ht_CAN4_ADDB_Tx.ID		:=	16#18200BDD OR EPEC_CANVXD.MASK_29BIT;
ht_CAN4_ADDB_Tx.Data[0]	:=	OrionBMS2_Rx.OrionBMS2_6BB_Rx.au8_Data[0];
ht_CAN4_ADDB_Tx.Data[1]	:=	OrionBMS2_Rx.OrionBMS2_6BB_Rx.au8_Data[1];
ht_CAN4_ADDB_Tx.Data[2]	:=	OrionBMS2_Rx.OrionBMS2_6BB_Rx.au8_Data[2];
ht_CAN4_ADDB_Tx.Data[3]	:=	OrionBMS2_Rx.OrionBMS2_6BB_Rx.au8_Data[3];
ht_CAN4_ADDB_Tx.Data[4]	:=	OrionBMS2_Rx.OrionBMS2_6BB_Rx.au8_Data[4];
ht_CAN4_ADDB_Tx.Data[5]	:=	OrionBMS2_Rx.OrionBMS2_6BB_Rx.au8_Data[5];		
ht_CAN4_ADDB_Tx.Data[6]	:=	OrionBMS2_Rx.OrionBMS2_6BB_Rx.au8_Data[6];	
ht_CAN4_ADDB_Tx.Data[7]	:=	OrionBMS2_Rx.OrionBMS2_6BB_Rx.au8_Data[7];		
ht_CAN4_ADDB_Tx.Len		:=	8;

ht_CAN4_ADDC_Tx.ID		:=	16#18200CDD OR EPEC_CANVXD.MASK_29BIT;
ht_CAN4_ADDC_Tx.Data[0]	:=	OrionBMS2_Rx.OrionBMS2_6BC_Rx.au8_Data[0];
ht_CAN4_ADDC_Tx.Data[1]	:=	OrionBMS2_Rx.OrionBMS2_6BC_Rx.au8_Data[1];
ht_CAN4_ADDC_Tx.Data[2]	:=	OrionBMS2_Rx.OrionBMS2_6BC_Rx.au8_Data[2];
ht_CAN4_ADDC_Tx.Data[3]	:=	OrionBMS2_Rx.OrionBMS2_6BC_Rx.au8_Data[3];
ht_CAN4_ADDC_Tx.Data[4]	:=	OrionBMS2_Rx.OrionBMS2_6BC_Rx.au8_Data[4];
ht_CAN4_ADDC_Tx.Data[5]	:=	OrionBMS2_Rx.OrionBMS2_6BC_Rx.au8_Data[5];		
ht_CAN4_ADDC_Tx.Data[6]	:=	OrionBMS2_Rx.OrionBMS2_6BC_Rx.au8_Data[6];	
ht_CAN4_ADDC_Tx.Data[7]	:=	OrionBMS2_Rx.OrionBMS2_6BC_Rx.au8_Data[7];		
ht_CAN4_ADDC_Tx.Len		:=	8;

ht_CAN4_ADDD_Tx.ID		:=	16#18200DDD OR EPEC_CANVXD.MASK_29BIT;
ht_CAN4_ADDD_Tx.Data[0]	:=	OrionBMS2_Rx.OrionBMS2_6BD_Rx.au8_Data[0];
ht_CAN4_ADDD_Tx.Data[1]	:=	OrionBMS2_Rx.OrionBMS2_6BD_Rx.au8_Data[1];
ht_CAN4_ADDD_Tx.Data[2]	:=	OrionBMS2_Rx.OrionBMS2_6BD_Rx.au8_Data[2];
ht_CAN4_ADDD_Tx.Data[3]	:=	OrionBMS2_Rx.OrionBMS2_6BD_Rx.au8_Data[3];
ht_CAN4_ADDD_Tx.Data[4]	:=	OrionBMS2_Rx.OrionBMS2_6BD_Rx.au8_Data[4];
ht_CAN4_ADDD_Tx.Data[5]	:=	OrionBMS2_Rx.OrionBMS2_6BD_Rx.au8_Data[5];		
ht_CAN4_ADDD_Tx.Data[6]	:=	OrionBMS2_Rx.OrionBMS2_6BD_Rx.au8_Data[6];	
ht_CAN4_ADDD_Tx.Data[7]	:=	OrionBMS2_Rx.OrionBMS2_6BD_Rx.au8_Data[7];		
ht_CAN4_ADDD_Tx.Len		:=	8;



Tx_Timer(IN := NOT(Tx_Timer.Q), PT := T#1000MS);
IF (Tx_Timer.Q = TRUE) THEN
	G_CAN4_Channel.SendMessage(i_pMSG:=ADR(ht_CAN4_DD0_Tx));
	G_CAN4_Channel.SendMessage(i_pMSG:=ADR(ht_CAN4_DD1_Tx));
	G_CAN4_Channel.SendMessage(i_pMSG:=ADR(ht_CAN4_DD2_Tx));
	G_CAN4_Channel.SendMessage(i_pMSG:=ADR(ht_CAN4_DD3_Tx));
	G_CAN4_Channel.SendMessage(i_pMSG:=ADR(ht_CAN4_DD4_Tx));
	G_CAN4_Channel.SendMessage(i_pMSG:=ADR(ht_CAN4_DD5_Tx));
	G_CAN4_Channel.SendMessage(i_pMSG:=ADR(ht_CAN4_DD6_Tx));
	G_CAN4_Channel.SendMessage(i_pMSG:=ADR(ht_CAN4_DD7_Tx));
	G_CAN4_Channel.SendMessage(i_pMSG:=ADR(ht_CAN4_DD8_Tx));
	G_CAN4_Channel.SendMessage(i_pMSG:=ADR(ht_CAN4_DD9_Tx));
	G_CAN4_Channel.SendMessage(i_pMSG:=ADR(ht_CAN4_DDA_Tx));
	G_CAN4_Channel.SendMessage(i_pMSG:=ADR(ht_CAN4_DDB_Tx));
	G_CAN4_Channel.SendMessage(i_pMSG:=ADR(ht_CAN4_DDC_Tx));
	G_CAN4_Channel.SendMessage(i_pMSG:=ADR(ht_CAN4_DDD_Tx));
	G_CAN4_Channel.SendMessage(i_pMSG:=ADR(ht_CAN4_ADD0_Tx));
	G_CAN4_Channel.SendMessage(i_pMSG:=ADR(ht_CAN4_ADD1_Tx));
	G_CAN4_Channel.SendMessage(i_pMSG:=ADR(ht_CAN4_ADD2_Tx));
	G_CAN4_Channel.SendMessage(i_pMSG:=ADR(ht_CAN4_ADD3_Tx));
	G_CAN4_Channel.SendMessage(i_pMSG:=ADR(ht_CAN4_ADD4_Tx));
	G_CAN4_Channel.SendMessage(i_pMSG:=ADR(ht_CAN4_ADD5_Tx));
	G_CAN4_Channel.SendMessage(i_pMSG:=ADR(ht_CAN4_ADD6_Tx));
	G_CAN4_Channel.SendMessage(i_pMSG:=ADR(ht_CAN4_ADD7_Tx));
	G_CAN4_Channel.SendMessage(i_pMSG:=ADR(ht_CAN4_ADD8_Tx));
	G_CAN4_Channel.SendMessage(i_pMSG:=ADR(ht_CAN4_ADD9_Tx));
	G_CAN4_Channel.SendMessage(i_pMSG:=ADR(ht_CAN4_ADDA_Tx));
	G_CAN4_Channel.SendMessage(i_pMSG:=ADR(ht_CAN4_ADDB_Tx));
	G_CAN4_Channel.SendMessage(i_pMSG:=ADR(ht_CAN4_ADDC_Tx));
	G_CAN4_Channel.SendMessage(i_pMSG:=ADR(ht_CAN4_ADDD_Tx));
	
END_IF

END_PROGRAM

// Application/UserCode/CAN4/Data to or For HMI/DCDC_to_HMI
PROGRAM DCDC_to_HMI
VAR
	ht_CAN4_5DD0_Tx	:	EPEC_CANVXD.Msg;
	ht_CAN4_5DD1_Tx: 	EPEC_CANVXD.Msg;
	hton_MessageSend_Timer	:	TON;
	
	Tx_Timer	:	TON;
	
END_VAR


//DCDC
ht_CAN4_5DD0_Tx.ID		:=	16#185000DD OR EPEC_CANVXD.MASK_29BIT;
ht_CAN4_5DD0_Tx.Data[0]	:=	BELDCDC_Rx.BelDCDC_IO_Rx.au8_Data[0];
ht_CAN4_5DD0_Tx.Data[1]	:=	BELDCDC_Rx.BelDCDC_IO_Rx.au8_Data[1];
ht_CAN4_5DD0_Tx.Data[2]	:=	BELDCDC_Rx.BelDCDC_IO_Rx.au8_Data[2];
ht_CAN4_5DD0_Tx.Data[3]	:=	BELDCDC_Rx.BelDCDC_IO_Rx.au8_Data[3];
ht_CAN4_5DD0_Tx.Data[4]	:=	BELDCDC_Rx.BelDCDC_IO_Rx.au8_Data[4];
ht_CAN4_5DD0_Tx.Data[5]	:=	BELDCDC_Rx.BelDCDC_IO_Rx.au8_Data[5];	
ht_CAN4_5DD0_Tx.Data[6]	:=	BELDCDC_Rx.BelDCDC_IO_Rx.au8_Data[6];	
ht_CAN4_5DD0_Tx.Data[7]	:=	BELDCDC_Rx.BelDCDC_IO_Rx.au8_Data[7];	
ht_CAN4_5DD0_Tx.Len		:=	8;

ht_CAN4_5DD1_Tx.ID		:=	16#185001DD OR EPEC_CANVXD.MASK_29BIT;
ht_CAN4_5DD1_Tx.Data[0]	:=	BELDCDC_Rx.BelDCDC_FWS_Rx.au8_Data[0];
ht_CAN4_5DD1_Tx.Data[1]	:=	BELDCDC_Rx.BelDCDC_FWS_Rx.au8_Data[1];
ht_CAN4_5DD1_Tx.Data[2]	:=	BELDCDC_Rx.BelDCDC_FWS_Rx.au8_Data[2];
ht_CAN4_5DD1_Tx.Data[3]	:=	BELDCDC_Rx.BelDCDC_FWS_Rx.au8_Data[3];
ht_CAN4_5DD1_Tx.Data[4]	:=	BELDCDC_Rx.BelDCDC_FWS_Rx.au8_Data[4];
ht_CAN4_5DD1_Tx.Data[5]	:=	BELDCDC_Rx.BelDCDC_FWS_Rx.au8_Data[5];	
ht_CAN4_5DD1_Tx.Data[6]	:=	BELDCDC_Rx.BelDCDC_FWS_Rx.au8_Data[6];	
ht_CAN4_5DD1_Tx.Data[7]	:=	BELDCDC_Rx.BelDCDC_FWS_Rx.au8_Data[7];	
ht_CAN4_5DD1_Tx.Len		:=	8;


Tx_Timer(IN := NOT(Tx_Timer.Q), PT := T#1000MS);
IF (Tx_Timer.Q = TRUE) THEN
	G_CAN4_Channel.SendMessage(i_pMSG:=ADR(ht_CAN4_5DD0_Tx));
	G_CAN4_Channel.SendMessage(i_pMSG:=ADR(ht_CAN4_5DD1_Tx));
	
	END_IF

END_PROGRAM

// Application/UserCode/CAN4/Data to or For HMI/MCU_to_HMI
PROGRAM MCU_to_HMI
VAR
	ht_CAN4_6DD0_Tx	:	EPEC_CANVXD.Msg;
	ht_CAN4_6DD1_Tx	:	EPEC_CANVXD.Msg;
	ht_CAN4_6DD2_Tx	:	EPEC_CANVXD.Msg;
	ht_CAN4_6DD3_Tx: EPEC_CANVXD.Msg;
	ht_CAN4_6DD4_Tx: EPEC_CANVXD.Msg;
	ht_CAN4_6DD5_Tx: EPEC_CANVXD.Msg;
	ht_CAN4_6DD6_Tx: EPEC_CANVXD.Msg;
	ht_CAN4_6DD7_Tx: EPEC_CANVXD.Msg;
	ht_CAN4_6DD8_Tx: EPEC_CANVXD.Msg;
	hton_MessageSend_Timer	:	TON;
	
	Tx_Timer	:	TON;
	
END_VAR


//MCU
ht_CAN4_6DD0_Tx.ID		:=	16#186000DD OR EPEC_CANVXD.MASK_29BIT;
ht_CAN4_6DD0_Tx.Data[0]	:=	MCU_Rx.MCU_Info1_Rx.au8_Data[0];
ht_CAN4_6DD0_Tx.Data[1]	:=	MCU_Rx.MCU_Info1_Rx.au8_Data[1];
ht_CAN4_6DD0_Tx.Data[2]	:=	MCU_Rx.MCU_Info1_Rx.au8_Data[2];
ht_CAN4_6DD0_Tx.Data[3]	:=	MCU_Rx.MCU_Info1_Rx.au8_Data[3];
ht_CAN4_6DD0_Tx.Data[4]	:=	MCU_Rx.MCU_Info1_Rx.au8_Data[4];
ht_CAN4_6DD0_Tx.Data[5]	:=	MCU_Rx.MCU_Info1_Rx.au8_Data[5];
ht_CAN4_6DD0_Tx.Data[6]	:=	MCU_Rx.MCU_Info1_Rx.au8_Data[6];
ht_CAN4_6DD0_Tx.Data[7]	:=	MCU_Rx.MCU_Info1_Rx.au8_Data[7];
ht_CAN4_6DD0_Tx.Len		:=	8;

ht_CAN4_6DD1_Tx.ID		:=	16#186001DD OR EPEC_CANVXD.MASK_29BIT;
ht_CAN4_6DD1_Tx.Data[0]	:=	MCU_Rx.MCU_Info2_Rx.au8_Data[0];
ht_CAN4_6DD1_Tx.Data[1]	:=	MCU_Rx.MCU_Info2_Rx.au8_Data[1];
ht_CAN4_6DD1_Tx.Data[2]	:=	MCU_Rx.MCU_Info2_Rx.au8_Data[2];
ht_CAN4_6DD1_Tx.Data[3]	:=	MCU_Rx.MCU_Info2_Rx.au8_Data[3];
ht_CAN4_6DD1_Tx.Data[4]	:=	MCU_Rx.MCU_Info2_Rx.au8_Data[4];
ht_CAN4_6DD1_Tx.Data[5]	:=	MCU_Rx.MCU_Info2_Rx.au8_Data[5];
ht_CAN4_6DD1_Tx.Data[6]	:=	MCU_Rx.MCU_Info2_Rx.au8_Data[6];
ht_CAN4_6DD1_Tx.Data[7]	:=	MCU_Rx.MCU_Info2_Rx.au8_Data[7];
ht_CAN4_6DD1_Tx.Len		:=	8;

ht_CAN4_6DD2_Tx.ID		:=	16#186002DD OR EPEC_CANVXD.MASK_29BIT;
ht_CAN4_6DD2_Tx.Data[0]	:=	MCU_Tx.ht_MCU_VMUComm1_Tx.Data[0];
ht_CAN4_6DD2_Tx.Data[1]	:=	MCU_Tx.ht_MCU_VMUComm1_Tx.Data[1];
ht_CAN4_6DD2_Tx.Data[2]	:=	MCU_Tx.ht_MCU_VMUComm1_Tx.Data[2];
ht_CAN4_6DD2_Tx.Data[3]	:=	MCU_Tx.ht_MCU_VMUComm1_Tx.Data[3];
ht_CAN4_6DD2_Tx.Data[4]	:=	MCU_Tx.ht_MCU_VMUComm1_Tx.Data[4];
ht_CAN4_6DD2_Tx.Data[5]	:=	MCU_Tx.ht_MCU_VMUComm1_Tx.Data[5];
ht_CAN4_6DD2_Tx.Data[6]	:=	MCU_Tx.ht_MCU_VMUComm1_Tx.Data[6];
ht_CAN4_6DD2_Tx.Data[7]	:=	MCU_Tx.ht_MCU_VMUComm1_Tx.Data[7];
ht_CAN4_6DD2_Tx.Len		:=	8;

ht_CAN4_6DD3_Tx.ID		:=	16#186003DD OR EPEC_CANVXD.MASK_29BIT;
ht_CAN4_6DD3_Tx.Data[0]	:=	MCU_Tx.ht_MCU_VMUComm2_Tx.Data[0];
ht_CAN4_6DD3_Tx.Data[1]	:=	MCU_Tx.ht_MCU_VMUComm2_Tx.Data[1];
ht_CAN4_6DD3_Tx.Data[2]	:=	MCU_Tx.ht_MCU_VMUComm2_Tx.Data[2];
ht_CAN4_6DD3_Tx.Data[3]	:=	MCU_Tx.ht_MCU_VMUComm2_Tx.Data[3];
ht_CAN4_6DD3_Tx.Data[4]	:=	MCU_Tx.ht_MCU_VMUComm2_Tx.Data[4];
ht_CAN4_6DD3_Tx.Data[5]	:=	MCU_Tx.ht_MCU_VMUComm2_Tx.Data[5];
ht_CAN4_6DD3_Tx.Data[6]	:=	MCU_Tx.ht_MCU_VMUComm2_Tx.Data[6];
ht_CAN4_6DD3_Tx.Data[7]	:=	MCU_Tx.ht_MCU_VMUComm2_Tx.Data[7];
ht_CAN4_6DD3_Tx.Len		:=	8;

ht_CAN4_6DD5_Tx.ID		:=	16#186005DD OR EPEC_CANVXD.MASK_29BIT;
ht_CAN4_6DD5_Tx.Data[0]	:=	MCU_Rx.MCU_CommandResponse1_Rx.au8_Data[0];
ht_CAN4_6DD5_Tx.Data[1]	:=	MCU_Rx.MCU_CommandResponse1_Rx.au8_Data[1];
ht_CAN4_6DD5_Tx.Data[2]	:=	MCU_Rx.MCU_CommandResponse1_Rx.au8_Data[2];
ht_CAN4_6DD5_Tx.Data[3]	:=	MCU_Rx.MCU_CommandResponse1_Rx.au8_Data[3];
ht_CAN4_6DD5_Tx.Data[4]	:=	MCU_Rx.MCU_CommandResponse1_Rx.au8_Data[4];
ht_CAN4_6DD5_Tx.Data[5]	:=	MCU_Rx.MCU_CommandResponse1_Rx.au8_Data[5];
ht_CAN4_6DD5_Tx.Data[6]	:=	MCU_Rx.MCU_CommandResponse1_Rx.au8_Data[6];
ht_CAN4_6DD5_Tx.Data[7]	:=	MCU_Rx.MCU_CommandResponse1_Rx.au8_Data[7];
ht_CAN4_6DD5_Tx.Len		:=	8;

ht_CAN4_6DD6_Tx.ID		:=	16#186006DD OR EPEC_CANVXD.MASK_29BIT;
ht_CAN4_6DD6_Tx.Data[0]	:=	MCU_Rx.MCU_CommandResponse2_Rx.au8_Data[0];
ht_CAN4_6DD6_Tx.Data[1]	:=	MCU_Rx.MCU_CommandResponse2_Rx.au8_Data[1];
ht_CAN4_6DD6_Tx.Data[2]	:=	MCU_Rx.MCU_CommandResponse2_Rx.au8_Data[2];
ht_CAN4_6DD6_Tx.Data[3]	:=	MCU_Rx.MCU_CommandResponse2_Rx.au8_Data[3];
ht_CAN4_6DD6_Tx.Data[4]	:=	MCU_Rx.MCU_CommandResponse2_Rx.au8_Data[4];
ht_CAN4_6DD6_Tx.Data[5]	:=	MCU_Rx.MCU_CommandResponse2_Rx.au8_Data[5];
ht_CAN4_6DD6_Tx.Data[6]	:=	MCU_Rx.MCU_CommandResponse2_Rx.au8_Data[6];
ht_CAN4_6DD6_Tx.Data[7]	:=	MCU_Rx.MCU_CommandResponse2_Rx.au8_Data[7];
ht_CAN4_6DD6_Tx.Len		:=	8;

ht_CAN4_6DD7_Tx.ID		:=	16#186007DD OR EPEC_CANVXD.MASK_29BIT;
ht_CAN4_6DD7_Tx.Data[0]	:=	MCU_Rx.MCU_EventInfo1_Rx.au8_Data[0];
ht_CAN4_6DD7_Tx.Data[1]	:=	MCU_Rx.MCU_EventInfo1_Rx.au8_Data[1];
ht_CAN4_6DD7_Tx.Data[2]	:=	MCU_Rx.MCU_EventInfo1_Rx.au8_Data[2];
ht_CAN4_6DD7_Tx.Data[3]	:=	MCU_Rx.MCU_EventInfo1_Rx.au8_Data[3];
ht_CAN4_6DD7_Tx.Data[4]	:=	MCU_Rx.MCU_EventInfo1_Rx.au8_Data[4];
ht_CAN4_6DD7_Tx.Data[5]	:=	MCU_Rx.MCU_EventInfo1_Rx.au8_Data[5];
ht_CAN4_6DD7_Tx.Data[6]	:=	MCU_Rx.MCU_EventInfo1_Rx.au8_Data[6];
ht_CAN4_6DD7_Tx.Data[7]	:=	MCU_Rx.MCU_EventInfo1_Rx.au8_Data[7];
ht_CAN4_6DD7_Tx.Len		:=	8;

ht_CAN4_6DD8_Tx.ID		:=	16#186008DD OR EPEC_CANVXD.MASK_29BIT;
ht_CAN4_6DD8_Tx.Data[0]	:=	MCU_Rx.MCU_Thermal1_Rx.au8_Data[0];
ht_CAN4_6DD8_Tx.Data[1]	:=	MCU_Rx.MCU_Thermal1_Rx.au8_Data[1];
ht_CAN4_6DD8_Tx.Data[2]	:=	MCU_Rx.MCU_Thermal1_Rx.au8_Data[2];
ht_CAN4_6DD8_Tx.Data[3]	:=	MCU_Rx.MCU_Thermal1_Rx.au8_Data[3];
ht_CAN4_6DD8_Tx.Data[4]	:=	MCU_Rx.MCU_Thermal1_Rx.au8_Data[4];
ht_CAN4_6DD8_Tx.Data[5]	:=	MCU_Rx.MCU_Thermal1_Rx.au8_Data[5];
ht_CAN4_6DD8_Tx.Data[6]	:=	MCU_Rx.MCU_Thermal1_Rx.au8_Data[6];
ht_CAN4_6DD8_Tx.Data[7]	:=	MCU_Rx.MCU_Thermal1_Rx.au8_Data[7];
ht_CAN4_6DD8_Tx.Len		:=	8;


Tx_Timer(IN := NOT(Tx_Timer.Q), PT := T#1000MS);
IF (Tx_Timer.Q = TRUE) THEN
	
	G_CAN4_Channel.SendMessage(i_pMSG:=ADR(ht_CAN4_6DD0_Tx));
	G_CAN4_Channel.SendMessage(i_pMSG:=ADR(ht_CAN4_6DD1_Tx));
	G_CAN4_Channel.SendMessage(i_pMSG:=ADR(ht_CAN4_6DD2_Tx));
	G_CAN4_Channel.SendMessage(i_pMSG:=ADR(ht_CAN4_6DD3_Tx));
	G_CAN4_Channel.SendMessage(i_pMSG:=ADR(ht_CAN4_6DD4_Tx));
	G_CAN4_Channel.SendMessage(i_pMSG:=ADR(ht_CAN4_6DD5_Tx));
	G_CAN4_Channel.SendMessage(i_pMSG:=ADR(ht_CAN4_6DD6_Tx));
	G_CAN4_Channel.SendMessage(i_pMSG:=ADR(ht_CAN4_6DD7_Tx));
	G_CAN4_Channel.SendMessage(i_pMSG:=ADR(ht_CAN4_6DD8_Tx));
	END_IF

END_PROGRAM

// Application/UserCode/CAN4/Data to or For HMI/Sevcon_to_HMI
PROGRAM Sevcon_to_HMI
VAR
	ht_CAN4_3DD0_Tx	:	EPEC_CANVXD.Msg;
	ht_CAN4_3DD1_Tx	:	EPEC_CANVXD.Msg;
	ht_CAN4_3DD2_Tx	:	EPEC_CANVXD.Msg;
	ht_CAN4_4DD0_Tx	:	EPEC_CANVXD.Msg;
	ht_CAN4_4DD1_Tx	:	EPEC_CANVXD.Msg;
	ht_CAN4_4DD2_Tx	:	EPEC_CANVXD.Msg;
	ht_CAN4_4DD3_Tx	:	EPEC_CANVXD.Msg;
	hton_MessageSend_Timer	:	TON;
	
	Tx_Timer	:	TON;
END_VAR


//*PowerSteering SEVCON
ht_CAN4_3DD0_Tx.ID		:=	16#183000DD OR EPEC_CANVXD.MASK_29BIT;
ht_CAN4_3DD0_Tx.Data[0]	:=	Sevcon_Steer_Rx.TorqueStatus1_Rx.au8_Data[0];
ht_CAN4_3DD0_Tx.Data[1]	:=	Sevcon_Steer_Rx.TorqueStatus1_Rx.au8_Data[1];
ht_CAN4_3DD0_Tx.Data[2]	:=	Sevcon_Steer_Rx.TorqueStatus1_Rx.au8_Data[2];
ht_CAN4_3DD0_Tx.Data[3]	:=	Sevcon_Steer_Rx.TorqueStatus1_Rx.au8_Data[3];
ht_CAN4_3DD0_Tx.Data[4]	:=	Sevcon_Steer_Rx.TorqueStatus1_Rx.au8_Data[4];
ht_CAN4_3DD0_Tx.Data[5]	:=	Sevcon_Steer_Rx.TorqueStatus1_Rx.au8_Data[5];
ht_CAN4_3DD0_Tx.Data[6]	:=	Sevcon_Steer_Rx.TorqueStatus1_Rx.au8_Data[6];
ht_CAN4_3DD0_Tx.Data[7]	:=	Sevcon_Steer_Rx.TorqueStatus1_Rx.au8_Data[7];
ht_CAN4_3DD0_Tx.Len		:=	8;

ht_CAN4_3DD1_Tx.ID		:=	16#183001DD OR EPEC_CANVXD.MASK_29BIT;
ht_CAN4_3DD1_Tx.Data[0]	:=	Sevcon_Steer_Rx.TorqueStatus2_Rx.au8_Data[0];
ht_CAN4_3DD1_Tx.Data[1]	:=	Sevcon_Steer_Rx.TorqueStatus2_Rx.au8_Data[1];
ht_CAN4_3DD1_Tx.Data[2]	:=	Sevcon_Steer_Rx.TorqueStatus2_Rx.au8_Data[2];
ht_CAN4_3DD1_Tx.Data[3]	:=	Sevcon_Steer_Rx.TorqueStatus2_Rx.au8_Data[3];
ht_CAN4_3DD1_Tx.Data[4]	:=	Sevcon_Steer_Rx.TorqueStatus2_Rx.au8_Data[4];
ht_CAN4_3DD1_Tx.Data[5]	:=	Sevcon_Steer_Rx.TorqueStatus2_Rx.au8_Data[5];
ht_CAN4_3DD1_Tx.Data[6]	:=	Sevcon_Steer_Rx.TorqueStatus2_Rx.au8_Data[6];
ht_CAN4_3DD1_Tx.Data[7]	:=	Sevcon_Steer_Rx.TorqueStatus2_Rx.au8_Data[7];
ht_CAN4_3DD1_Tx.Len		:=	8;

ht_CAN4_3DD2_Tx.ID		:=	16#183002DD OR EPEC_CANVXD.MASK_29BIT;
ht_CAN4_3DD2_Tx.Data[0]	:=	Sevcon_Steer_Rx.TempStatus_Rx.au8_Data[0];
ht_CAN4_3DD2_Tx.Data[1]	:=	Sevcon_Steer_Rx.TempStatus_Rx.au8_Data[1];
ht_CAN4_3DD2_Tx.Data[2]	:=	gu8_Sevcon1_Debug_Temp_Heatsink;
ht_CAN4_3DD2_Tx.Data[3]	:=	Sevcon_Steer_Rx.TempStatus_Rx.au8_Data[3];
ht_CAN4_3DD2_Tx.Data[4]	:=	Sevcon_Steer_Rx.TempStatus_Rx.au8_Data[4];
ht_CAN4_3DD2_Tx.Data[5]	:=	Sevcon_Steer_Rx.TempStatus_Rx.au8_Data[5];
ht_CAN4_3DD2_Tx.Data[6]	:=	Sevcon_Steer_Rx.TempStatus_Rx.au8_Data[6];
ht_CAN4_3DD2_Tx.Data[7]	:=	Sevcon_Steer_Rx.TempStatus_Rx.au8_Data[7];
ht_CAN4_3DD2_Tx.Len		:=	8;

(*Compressor SEVCON*)
ht_CAN4_4DD0_Tx.ID		:=	16#184000DD OR EPEC_CANVXD.MASK_29BIT;
ht_CAN4_4DD0_Tx.Data[0]	:=	Sevcon2_Rx.TorqueStatus1_Rx.au8_Data[0];
ht_CAN4_4DD0_Tx.Data[1]	:=	Sevcon2_Rx.TorqueStatus1_Rx.au8_Data[1];
ht_CAN4_4DD0_Tx.Data[2]	:=	Sevcon2_Rx.TorqueStatus1_Rx.au8_Data[2];
ht_CAN4_4DD0_Tx.Data[3]	:=	Sevcon2_Rx.TorqueStatus1_Rx.au8_Data[3];
ht_CAN4_4DD0_Tx.Data[4]	:=	Sevcon2_Rx.TorqueStatus1_Rx.au8_Data[4];
ht_CAN4_4DD0_Tx.Data[5]	:=	Sevcon2_Rx.TorqueStatus1_Rx.au8_Data[5];
ht_CAN4_4DD0_Tx.Data[6]	:=	Sevcon2_Rx.TorqueStatus1_Rx.au8_Data[6];
ht_CAN4_4DD0_Tx.Data[7]	:=	Sevcon2_Rx.TorqueStatus1_Rx.au8_Data[7];
ht_CAN4_4DD0_Tx.Len		:=	8;

ht_CAN4_4DD1_Tx.ID		:=	16#184001DD OR EPEC_CANVXD.MASK_29BIT;
ht_CAN4_4DD1_Tx.Data[0]	:=	Sevcon2_Rx.TorqueStatus2_Rx.au8_Data[0];
ht_CAN4_4DD1_Tx.Data[1]	:=	Sevcon2_Rx.TorqueStatus2_Rx.au8_Data[1];
ht_CAN4_4DD1_Tx.Data[2]	:=	Sevcon2_Rx.TorqueStatus2_Rx.au8_Data[2];
ht_CAN4_4DD1_Tx.Data[3]	:=	Sevcon2_Rx.TorqueStatus2_Rx.au8_Data[3];
ht_CAN4_4DD1_Tx.Data[4]	:=	Sevcon2_Rx.TorqueStatus2_Rx.au8_Data[4];
ht_CAN4_4DD1_Tx.Data[5]	:=	Sevcon2_Rx.TorqueStatus2_Rx.au8_Data[5];
ht_CAN4_4DD1_Tx.Data[6]	:=	Sevcon2_Rx.TorqueStatus2_Rx.au8_Data[6];
ht_CAN4_4DD1_Tx.Data[7]	:=	Sevcon2_Rx.TorqueStatus2_Rx.au8_Data[7];
ht_CAN4_4DD1_Tx.Len		:=	8;

ht_CAN4_4DD2_Tx.ID		:=	16#184002DD OR EPEC_CANVXD.MASK_29BIT;
ht_CAN4_4DD2_Tx.Data[0]	:=	Sevcon2_Rx.TempStatus_Rx.au8_Data[0];
ht_CAN4_4DD2_Tx.Data[1]	:=	Sevcon2_Rx.TempStatus_Rx.au8_Data[1];
ht_CAN4_4DD2_Tx.Data[2]	:=	Sevcon2_Rx.TempStatus_Rx.au8_Data[2];
ht_CAN4_4DD2_Tx.Data[3]	:=	Sevcon2_Rx.TempStatus_Rx.au8_Data[3];
ht_CAN4_4DD2_Tx.Data[4]	:=	Sevcon2_Rx.TempStatus_Rx.au8_Data[4];
ht_CAN4_4DD2_Tx.Data[5]	:=	Sevcon2_Rx.TempStatus_Rx.au8_Data[5];
ht_CAN4_4DD2_Tx.Data[6]	:=	Sevcon2_Rx.TempStatus_Rx.au8_Data[6];
ht_CAN4_4DD2_Tx.Data[7]	:=	Sevcon2_Rx.TempStatus_Rx.au8_Data[7];
ht_CAN4_4DD2_Tx.Len		:=	8;

ht_CAN4_4DD3_Tx.ID		:=	16#184003DD OR EPEC_CANVXD.MASK_29BIT;
ht_CAN4_4DD3_Tx.Data[0]	:=	Sevcon2_Rx.Compressor_Temp_Rx.au8_Data[5];
ht_CAN4_4DD3_Tx.Data[1]	:=	Sevcon2_Rx.Compressor_Temp_Rx.au8_Data[6];
ht_CAN4_4DD3_Tx.Data[2]	:=	gu8_Sevcon1_Debug_Temp_Heatsink;
ht_CAN4_4DD3_Tx.Data[3].0	:= Sevcon2_Control.NO_OIL;
ht_CAN4_4DD3_Tx.Data[3].1	:= Sevcon2_Rx.Compressor_Oil_Rx.au8_Data[2].4;
ht_CAN4_4DD3_Tx.Data[3].2	:= Sevcon2_Control.Oil_Level_Warning;
ht_CAN4_4DD3_Tx.Data[3].3	:= Sevcon2_Control.Compressor_Temp_Warning;
ht_CAN4_4DD3_Tx.Data[3].4	:= Sevcon2_Control.Compressor_Temp_Fault;
ht_CAN4_4DD3_Tx.Data[3].5	:= Sevcon2_Control.Air_Temp_Warning;
ht_CAN4_4DD3_Tx.Data[3].6	:= Sevcon2_Control.Air_Temp_Fault;
ht_CAN4_4DD3_Tx.Data[3].7	:= CAN1_Rx.Bob_J1939_AirPressure_Rx.au8_Data[6].0;
ht_CAN4_4DD3_Tx.Data[4]	:=	16#00;
ht_CAN4_4DD3_Tx.Data[5]	:=	16#00;
ht_CAN4_4DD3_Tx.Data[6]	:=	16#00;
ht_CAN4_4DD3_Tx.Data[7]	:=	16#00;
ht_CAN4_4DD3_Tx.Len		:=	8;


Tx_Timer(IN := NOT(Tx_Timer.Q), PT := T#1000MS);
IF (Tx_Timer.Q = TRUE) THEN
	G_CAN4_Channel.SendMessage(i_pMSG:=ADR(ht_CAN4_3DD0_Tx));
	G_CAN4_Channel.SendMessage(i_pMSG:=ADR(ht_CAN4_3DD1_Tx));
	G_CAN4_Channel.SendMessage(i_pMSG:=ADR(ht_CAN4_3DD2_Tx));
	G_CAN4_Channel.SendMessage(i_pMSG:=ADR(ht_CAN4_4DD0_Tx));
	G_CAN4_Channel.SendMessage(i_pMSG:=ADR(ht_CAN4_4DD1_Tx));
	G_CAN4_Channel.SendMessage(i_pMSG:=ADR(ht_CAN4_4DD2_Tx));
	G_CAN4_Channel.SendMessage(i_pMSG:=ADR(ht_CAN4_4DD3_Tx));

END_IF

END_PROGRAM

// Application/UserCode/CAN4/Data to or For HMI/VMU_to_HMI
PROGRAM VMU_to_HMI
VAR
	CAN4_VMU0_Tx			:	EPEC_CANVXD.Msg;	// Digital
	CAN4_VMU1_Tx			: 	EPEC_CANVXD.Msg;	// Digital
	CAN4_VMU2_Tx			: 	EPEC_CANVXD.Msg;
	CAN4_VMU3_Tx			: 	EPEC_CANVXD.Msg;
	CAN4_VMU4_Tx			: 	EPEC_CANVXD.Msg;
	CAN4_VMU5_Tx			: 	EPEC_CANVXD.Msg;
	hton_MessageSend_Timer	:	TON;
	Tx_Timer				:	TON;
END_VAR

//called from can4_TX
// Connector C1 DIGITAL ONLY
CAN4_VMU0_Tx.ID			:=	16#190000DD OR EPEC_CANVXD.MASK_29BIT;
CAN4_VMU0_Tx.Len		:=	8;
CAN4_VMU0_Tx.Data[0].0	:= DI_q_BatteryInterlockIn_DI;					//Pin 1.11 - Filtered digital input status.
CAN4_VMU0_Tx.Data[0].1	:= DOS_q_BackupPump_DO;							//X1.12 Backup power steering
CAN4_VMU0_Tx.Data[0].2	:= DO_q_BackupPump_DO; 							//X1.12 Backup power steering
CAN4_VMU0_Tx.Data[0].3	:= DOS_q_BatteryDischargeMain_DO; 				//X1.22 Battery Discharge Main
CAN4_VMU0_Tx.Data[0].4	:= DO_q_BatteryDischargeMain_DO;  				//X1.22 Battery Discharge Main
CAN4_VMU0_Tx.Data[0].5	:= DOS_q_AirPressureReliefValve_DO; 			//X1.23 ePTO Fan Enable
CAN4_VMU0_Tx.Data[0].6	:= DO_q_AirPressureReliefValve_DO;				//X1.23 ePTO Fan Enable
CAN4_VMU0_Tx.Data[0].7  := DOS_q_Battery1ChargePrecharge_DO;			//X1.29 Soft Charge Battery 1
CAN4_VMU0_Tx.Data[1].0  := DO_q_Battery1ChargePrecharge_DO;				//X1.29 Soft Charge Battery 1
CAN4_VMU0_Tx.Data[1].1  := DOS_q_Battery1ChargeMain_DO; 				//X1.30 Charge Main Battery 1
CAN4_VMU0_Tx.Data[1].2  := DO_q_Battery1ChargeMain_DO;					//Pin 1.30 - Digital output status for output pin. 
CAN4_VMU0_Tx.Data[1].3  := DOS_q_Battery2ChargePrecharge_DO; 			//X1.31 Soft Charge Battery 2
CAN4_VMU0_Tx.Data[1].4  := DO_q_Battery2ChargePrecharge_DO;				//X1.31 Soft Charge Battery 2
CAN4_VMU0_Tx.Data[1].5  := DOS_q_DrivetrainInverterTorqueless_DO;		//Pin 1.32 - Digital input state for pin.	
CAN4_VMU0_Tx.Data[1].6  := DO_q_DrivetrainInverterTorqueless_DO;		//Pin 1.32 - Digital output status for output pin.
CAN4_VMU0_Tx.Data[1].7  := DOS_q_BatteryDischargePrecharge_DO; 			//X1.33 Soft Discharge Battery 1
CAN4_VMU0_Tx.Data[2].0  := DO_q_BatteryDischargePrecharge_DO;			//Pin 1.33 - Digital output status for output pin. 
CAN4_VMU0_Tx.Data[2].1  := DOS_q_Battery2ChargeMain_DO; 				//X1.35 Charge Main Battery 2
CAN4_VMU0_Tx.Data[2].2  := DO_q_Battery2ChargeMain_DO;					//Pin 1.35 - Digital output status for output pin.
// Connector C2 DIGITAL ONLY
CAN4_VMU0_Tx.Data[2].3  := DI_q_Battery1ChargeRq_DI; 					//Pin 2.6 - Filtered digital input status.
CAN4_VMU0_Tx.Data[2].4  := DI_q_Battery1DiscahrgeRq_DI; 				//Pin 2.7 - Filtered digital input status.
CAN4_VMU0_Tx.Data[2].5  := DI_q_Battery2ChargeRq_DI; 					//Pin 2.8 - Filtered digital input status.
CAN4_VMU0_Tx.Data[2].6  := DI_q_Batter2DischargeRq_DI; 					//Pin 2.9 - Filtered digital input status.
CAN4_VMU0_Tx.Data[2].7  := DOS_q_ChargePlugLockPulse_DO ; 				//Pin 2.13 - Digital input state for pin.
CAN4_VMU0_Tx.Data[3].0  := DO_q_ChargePlugLockPulse_DO;					//Pin 2.13 - Digital output status for output pin.
CAN4_VMU0_Tx.Data[3].1  := DOS_q_ChargePlugLockPosition_DO; 			//Pin 2.14 - Digital input state for pin.
CAN4_VMU0_Tx.Data[3].2  := DO_q_ChargePlugLockPosition_DO;				//Pin 2.14 - Digital output status for output pin.
CAN4_VMU0_Tx.Data[3].3  := DI_q_ChargePlugLockStatus_DI; 				//Pin 2.16 - Filtered digital input status.
CAN4_VMU0_Tx.Data[3].4  := DOS_q_DrivetrainKL15D_DO; 					//Pin 2.28 - Digital input state for pin.
CAN4_VMU0_Tx.Data[3].5  := DO_q_DrivetrainKL15D_DO;						//Pin 2.28 - Digital output status for output pin.
CAN4_VMU0_Tx.Data[3].6  := DOS_q_DrivetrainKL15C_DO; 					//Pin 2.29 - Digital input state for pin.
CAN4_VMU0_Tx.Data[3].7  := DO_q_DrivetrainKL15C_DO;						//Pin 2.29 - Digital output status for output pin.
CAN4_VMU0_Tx.Data[4].0  := DOS_q_DrivetrainCoolingFan_DO; 				//Pin 2.30 - Digital input state for pin.
CAN4_VMU0_Tx.Data[4].1  := DO_q_DrivetrainCoolingFan_DO;				//Pin 2.30 - Digital output status for output pin.
CAN4_VMU0_Tx.Data[4].2  := DOS_q_DrievtrainPowerSteering_DO; 			//Pin 2.31 - Digital input state for pin.
CAN4_VMU0_Tx.Data[4].3  := DO_q_DrievtrainPowerSteering_DO;				//Pin 2.31 - Digital output status for output pin.
CAN4_VMU0_Tx.Data[4].4  := DOS_q_DrievtrainAirCompressor_DO; 			//Pin 2.33 - Digital input state for pin.
CAN4_VMU0_Tx.Data[4].5  := DO_q_DrievtrainAirCompressor_DO;				//Pin 2.33 - Digital output status for output pin.
CAN4_VMU0_Tx.Data[4].6  := DOS_q_DynamoD_DO; 							//Pin 2.35 - Digital input state for pin.
CAN4_VMU0_Tx.Data[4].7  := DO_q_DynamoD_DO;								//Pin 2.35 - Digital output state for sinking digital output.
// Connector C3 DIGITAL ONLY
CAN4_VMU0_Tx.Data[5].0  := DI_q_DirectionSwitch_ReverseCrawl_DI; 		//Pin 3.5 - Filtered digital input status.
CAN4_VMU0_Tx.Data[5].1  := DI_q_DirectionSwitch_Drive_DI; 				//Pin 3.6 - Filtered digital input status.
CAN4_VMU0_Tx.Data[5].2  := DI_q_IlluminiationStatsus_DI; 				//Pin 3.7 - Filtered digital input status.
CAN4_VMU0_Tx.Data[5].3  := DI_q_DirectionSwitch_Reverse_DI; 			//Pin 3.8 - Filtered digital input status.
CAN4_VMU0_Tx.Data[5].4  := DI_q_DirectionSwitch_DriveCrawl_DI; 			//Pin 3.9 - Filtered digital input status.
CAN4_VMU0_Tx.Data[5].5  := DI_q_DirectionSwitch_Neutral_DI; 			//Pin 3.11 - Filtered digital input status.
CAN4_VMU0_Tx.Data[5].6  := DI_q_VehicleKL15_DI; 						//Pin 3.22 - Filtered digital input status.
CAN4_VMU0_Tx.Data[5].7  := DI_q_VehicleKL51_DI; 						//Pin 3.23 - Filtered digital input status.
CAN4_VMU0_Tx.Data[6].0  := DOS_q_ChargersWakeup_DO; 					//Pin 3.26 - Digital input state for pin.
CAN4_VMU0_Tx.Data[6].1  := DO_q_ChargersWakeup_DO;						//Pin 3.26 - Digital output status for output pin.
CAN4_VMU0_Tx.Data[6].2  := DOS_q_DashboardDCDCStatus_DO; 				//Pin 3.27 - Digital input state for pin.
CAN4_VMU0_Tx.Data[6].3  := DO_q_DashboardDCDCStatus_DO;					//Pin 3.27 - Digital output status for output pin.
CAN4_VMU0_Tx.Data[6].4  := DI_q_HeaterIn_DI; 							//Pin 3.28 - Filtered digital input status.
CAN4_VMU0_Tx.Data[6].5  := DOS_q_HeaterOut_DI; 							//Pin 3.29 - Digital input state for pin.
CAN4_VMU0_Tx.Data[6].6  := DO_q_HeaterOut_DI;							//Pin 3.29 - Digital output status for output pin.
CAN4_VMU0_Tx.Data[6].7  := DOS_q_DrivetrainInverterRf1_DO; 				//Pin 3.30 - Digital input state for pin.
CAN4_VMU0_Tx.Data[7].0  := DO_q_DrivetrainInverterRf1_DO;				//Pin 3.30 - Digital output status for output pin.	
CAN4_VMU0_Tx.Data[7].1  := DOS_q_DrivetrainInverterRf2_DO; 				//Pin 3.31 - Digital input state for pin.
CAN4_VMU0_Tx.Data[7].2  := DO_q_DrivetrainInverterRf2_DO;				//Pin 3.31 - Digital output status for output pin.
CAN4_VMU0_Tx.Data[7].3  := DOS_q_DrivetrainDCDCInhibit_DO; 				//Pin 3.32 - Digital input state for pin.
CAN4_VMU0_Tx.Data[7].4  := DO_q_DrivetrainDCDCInhibit_DO;				//Pin 3.32 - Digital output status for output pin.
CAN4_VMU0_Tx.Data[7].5  := DOS_q_ChargePlugLED_Green_DO; 				//Pin 3.33 - Digital input state for pin.
CAN4_VMU0_Tx.Data[7].6  := DO_q_ChargePlugLED_Green_DO;					//Pin 3.33 - Digital output status for output pin.
CAN4_VMU0_Tx.Data[7].7  := DOS_q_ChargePlugLED_Blue_DO; 				//Pin 3.34 - Digital input state for pin.

// Connector C3 DIGITAL ONLY Continued
CAN4_VMU1_Tx.ID			:=	16#190001DD OR EPEC_CANVXD.MASK_29BIT;
CAN4_VMU1_Tx.Len		:=	8;
CAN4_VMU1_Tx.Data[0].0  := DO_q_ChargePlugLED_Blue_DO;					//Pin 3.34 - Digital output status for output pin.
CAN4_VMU1_Tx.Data[0].1  := DOS_q_ChargePlugLED_Red_DO; 					//Pin 3.35 - Digital input state for pin.
CAN4_VMU1_Tx.Data[0].2  := DO_q_ChargePlugLED_Red_DO;					//Pin 3.35 - Digital output status for output pin.
CAN4_VMU1_Tx.Data[0].3  := 0;											//Spare.
//Ditto																	//Ditto.

//Anal Stuff
CAN4_VMU2_Tx.ID			:=	16#190002DD OR EPEC_CANVXD.MASK_29BIT;
CAN4_VMU2_Tx.Len		:=	8;
CAN4_VMU2_Tx.Data[0]	:=	WORD_TO_BYTE 	(AIPU_u16_DrivetrainTemp_AI);				//Pin 1.9 - Filtered AI value
CAN4_VMU2_Tx.Data[1]	:=	WORD_TO_BYTE 	(SHR (AIPU_u16_DrivetrainTemp_AI, 8));		//Pin 1.9 - Filtered AI value
CAN4_VMU2_Tx.Data[2]	:=	WORD_TO_BYTE 	(AI_u16_DrivetrainTemp_AI);					//Pin 1.9 - Filtered AI value
CAN4_VMU2_Tx.Data[3]	:=	WORD_TO_BYTE 	(SHR (AI_u16_DrivetrainTemp_AI, 8));		//Pin 1.9 - Filtered AI value
CAN4_VMU2_Tx.Data[4]	:=	WORD_TO_BYTE 	(AIPU_u16_ChargePlugPresent_AI);			//Pin 1.10 - Filtered AI value
CAN4_VMU2_Tx.Data[5]	:=	WORD_TO_BYTE 	(SHR (AIPU_u16_ChargePlugPresent_AI, 8)); 	//Pin 1.10 - Filtered AI value
CAN4_VMU2_Tx.Data[6]	:=	WORD_TO_BYTE 	(AI_u16_ChargePlugPresent_AI);				//Pin 1.10 - Filtered AI value
CAN4_VMU2_Tx.Data[7]	:=	WORD_TO_BYTE 	(SHR (AI_u16_ChargePlugPresent_AI, 8));		//Pin 1.10 - Filtered AI value

CAN4_VMU3_Tx.ID			:=	16#190003DD OR EPEC_CANVXD.MASK_29BIT;
CAN4_VMU3_Tx.Len		:=	8;
CAN4_VMU3_Tx.Data[0]	:=	WORD_TO_BYTE 	(AIPU_u16_Heater1Temperature_AI);			//Pin 1.20 - Filtered AI value
CAN4_VMU3_Tx.Data[1]	:=	WORD_TO_BYTE 	(SHR (AIPU_u16_Heater1Temperature_AI, 8));	//Pin 1.20 - Filtered AI value
CAN4_VMU3_Tx.Data[2]	:=	WORD_TO_BYTE 	(AI_u16_Heater1Temperature_AI);				//Pin 1.20 - Filtered AI value
CAN4_VMU3_Tx.Data[3]	:=	WORD_TO_BYTE 	(SHR (AI_u16_Heater1Temperature_AI, 8));	//Pin 1.20 - Filtered AI value
CAN4_VMU3_Tx.Data[4]	:=	WORD_TO_BYTE 	(AIPU_u16_Heater2Temperature_AI);			//Pin 1.21 - Filtered AI value
CAN4_VMU3_Tx.Data[5]	:=	WORD_TO_BYTE 	(SHR (AIPU_u16_Heater2Temperature_AI, 8));	//Pin 1.21 - Filtered AI value
CAN4_VMU3_Tx.Data[6]	:=	WORD_TO_BYTE 	(AI_u16_Heater2Temperature_AI);				//Pin 1.21 - Filtered AI value
CAN4_VMU3_Tx.Data[7]	:=	WORD_TO_BYTE 	(SHR (AI_u16_Heater2Temperature_AI, 8));	//Pin 1.21 - Filtered AI value

CAN4_VMU4_Tx.ID			:=	16#190004DD OR EPEC_CANVXD.MASK_29BIT;		
CAN4_VMU4_Tx.Len		:=	8;				
CAN4_VMU4_Tx.Data[0]	:=	WORD_TO_BYTE 	(AIPU_u16_HeaterDiagnose_AI);				//Pin 2.23 - Filtered AI value
CAN4_VMU4_Tx.Data[1]	:=	WORD_TO_BYTE 	(SHR (AIPU_u16_HeaterDiagnose_AI, 8));		//Pin 2.23 - Filtered AI value
CAN4_VMU4_Tx.Data[2]	:=	WORD_TO_BYTE 	(AI_u16_HeaterDiagnose_AI);					//Pin 2.23 - Filtered AI value
CAN4_VMU4_Tx.Data[3]	:=	WORD_TO_BYTE 	(SHR (AI_u16_HeaterDiagnose_AI, 8));		//Pin 2.23 - Filtered AI value
CAN4_VMU4_Tx.Data[4]	:=	WORD_TO_BYTE 	(AIPU_u16_HeaterDiagnose2_AI);				//Pin 3.14 - Filtered AI value
CAN4_VMU4_Tx.Data[5]	:=	WORD_TO_BYTE 	(SHR (AIPU_u16_HeaterDiagnose2_AI, 8));		//Pin 3.14 - Filtered AI value
CAN4_VMU4_Tx.Data[6]	:=	WORD_TO_BYTE 	(AI_u16_Heater1Temperature_AI);				//Pin 3.14 - Filtered AI value
CAN4_VMU4_Tx.Data[7]	:=	WORD_TO_BYTE 	(SHR (AI_u16_Heater1Temperature_AI, 8));	//Pin 3.14 - Filtered AI value

CAN4_VMU5_Tx.ID			:=	16#190005DD OR EPEC_CANVXD.MASK_29BIT;
CAN4_VMU5_Tx.Len		:=	8;
CAN4_VMU5_Tx.Data[0]	:=	WORD_TO_BYTE 	(AIPU_u16_VehicleThrottlePedal1_AI);		//Pin 3.15 - Filtered AI value
CAN4_VMU5_Tx.Data[1]	:=	WORD_TO_BYTE 	(SHR(AIPU_u16_VehicleThrottlePedal1_AI,8)); //Pin 3.15 - Filtered AI value
CAN4_VMU5_Tx.Data[2]	:=	WORD_TO_BYTE 	(AI_u16_VehicleThrottlePedal1_AI);			//Pin 3.15 - Filtered AI value
CAN4_VMU5_Tx.Data[3]	:=	WORD_TO_BYTE 	(SHR (AI_u16_VehicleThrottlePedal1_AI,8));	//Pin 3.15 - Filtered AI value
CAN4_VMU5_Tx.Data[4]	:=	WORD_TO_BYTE 	(AIPU_u16_VehicleThrottlePedal2_AI	);		//Pin 3.16 - Filtered AI value 
CAN4_VMU5_Tx.Data[5]	:=	WORD_TO_BYTE 	(SHR(AIPU_u16_VehicleThrottlePedal2_AI,8)); //Pin 3.16 - Filtered AI value 
CAN4_VMU5_Tx.Data[6]	:=	WORD_TO_BYTE 	(AI_u16_VehicleThrottlePedal2_AI);			//Pin 3.16 - Filtered AI value 
CAN4_VMU5_Tx.Data[7]	:=	WORD_TO_BYTE 	(SHR(AI_u16_VehicleThrottlePedal2_AI, 8));	//Pin 3.16 - Filtered AI value 


Tx_Timer(IN := NOT(Tx_Timer.Q), PT := T#100MS);
IF (Tx_Timer.Q = TRUE) THEN
	G_CAN4_Channel.SendMessage(i_pMSG:=ADR(CAN4_VMU0_Tx));
	G_CAN4_Channel.SendMessage(i_pMSG:=ADR(CAN4_VMU1_Tx));
	G_CAN4_Channel.SendMessage(i_pMSG:=ADR(CAN4_VMU2_Tx));
	G_CAN4_Channel.SendMessage(i_pMSG:=ADR(CAN4_VMU3_Tx));
	G_CAN4_Channel.SendMessage(i_pMSG:=ADR(CAN4_VMU4_Tx));
	G_CAN4_Channel.SendMessage(i_pMSG:=ADR(CAN4_VMU5_Tx));
END_IF

END_PROGRAM

// Application/UserCode/CAN4/Data to or For HMI/BRUSA_to_HMI
PROGRAM BRUSA_to_HMI
VAR
	ht_CAN4_7DD0_Tx	:	EPEC_CANVXD.Msg;
	ht_CAN4_7DD1_Tx	:	EPEC_CANVXD.Msg;
	ht_CAN4_7DD2_Tx: EPEC_CANVXD.msg;
	ht_CAN4_7DD3_Tx: EPEC_CANVXD.msg;
	ht_CAN4_7DD4_Tx: EPEC_CANVXD.msg;
	ht_CAN4_7DD5_Tx: EPEC_CANVXD.msg;
	ht_CAN4_7DD6_Tx: EPEC_CANVXD.msg;
	ht_CAN4_7DD7_Tx: EPEC_CANVXD.msg;
	ht_CAN4_7DD8_Tx: EPEC_CANVXD.msg;
	ht_CAN4_7DD9_Tx: EPEC_CANVXD.msg;
	ht_CAN4_7DDA_Tx: EPEC_CANVXD.msg;
	ht_CAN4_7DDB_Tx: EPEC_CANVXD.msg;
	hton_MessageSend_Timer	:	TON;
	Tx_Timer	:	TON;
	END_VAR

//called from can4_TX

//Master Brusa
ht_CAN4_7DD0_Tx.ID		:=	16#187000DD OR EPEC_CANVXD.MASK_29BIT;
ht_CAN4_7DD0_Tx.Data[0]	:=	Brusa1_Rx.ActAC_Rx.au8_Data[0];
ht_CAN4_7DD0_Tx.Data[1]	:=	Brusa1_Rx.ActAC_Rx.au8_Data[1];
ht_CAN4_7DD0_Tx.Data[2]	:=	Brusa1_Rx.ActAC_Rx.au8_Data[2];
ht_CAN4_7DD0_Tx.Data[3]	:=	Brusa1_Rx.ActAC_Rx.au8_Data[3];
ht_CAN4_7DD0_Tx.Data[4]	:=	Brusa1_Rx.ActAC_Rx.au8_Data[4];
ht_CAN4_7DD0_Tx.Data[5]	:=	Brusa1_Rx.ActAC_Rx.au8_Data[5];
ht_CAN4_7DD0_Tx.Data[6]	:=	Brusa1_Rx.ActAC_Rx.au8_Data[6];
ht_CAN4_7DD0_Tx.Data[7]	:=	Brusa1_Rx.ActAC_Rx.au8_Data[7];
ht_CAN4_7DD0_Tx.Len		:=	8;

//* Errors
ht_CAN4_7DD2_Tx.ID		:=	16#187002DD OR EPEC_CANVXD.MASK_29BIT;
ht_CAN4_7DD2_Tx.Data[0]	:=	Brusa1_Rx.ActErr_Rx.au8_Data[0];
ht_CAN4_7DD2_Tx.Data[1]	:=	Brusa1_Rx.ActErr_Rx.au8_Data[1];
ht_CAN4_7DD2_Tx.Data[2]	:=	Brusa1_Rx.ActErr_Rx.au8_Data[2];
ht_CAN4_7DD2_Tx.Data[3]	:=	Brusa1_Rx.ActErr_Rx.au8_Data[3];
ht_CAN4_7DD2_Tx.Data[4]	:=	Brusa1_Rx.ActErr_Rx.au8_Data[4];
ht_CAN4_7DD2_Tx.Data[5]	:=	Brusa1_Rx.ActErr_Rx.au8_Data[5];
ht_CAN4_7DD2_Tx.Data[6]	:=	Brusa1_Rx.ActErr_Rx.au8_Data[6];
ht_CAN4_7DD2_Tx.Data[7]	:=	Brusa1_Rx.ActErr_Rx.au8_Data[7];
ht_CAN4_7DD2_Tx.Len		:=	8;

ht_CAN4_7DD4_Tx.ID		:=	16#187004DD OR EPEC_CANVXD.MASK_29BIT;
ht_CAN4_7DD4_Tx.Data[0]	:=	Brusa1_Rx.ActInt_Rx.au8_Data[0];
ht_CAN4_7DD4_Tx.Data[1]	:=	Brusa1_Rx.ActInt_Rx.au8_Data[1];
ht_CAN4_7DD4_Tx.Data[2]	:=	Brusa1_Rx.ActInt_Rx.au8_Data[2];
ht_CAN4_7DD4_Tx.Data[3]	:=	Brusa1_Rx.ActInt_Rx.au8_Data[3];
ht_CAN4_7DD4_Tx.Data[4]	:=	Brusa1_Rx.ActInt_Rx.au8_Data[4];
ht_CAN4_7DD4_Tx.Data[5]	:=	Brusa1_Rx.ActInt_Rx.au8_Data[5];
ht_CAN4_7DD4_Tx.Data[6]	:=	Brusa1_Rx.ActInt_Rx.au8_Data[6];
ht_CAN4_7DD4_Tx.Data[7]	:=	Brusa1_Rx.ActInt_Rx.au8_Data[7];
ht_CAN4_7DD4_Tx.Len		:=	8;

ht_CAN4_7DD6_Tx.ID		:=	16#187006DD OR EPEC_CANVXD.MASK_29BIT;
ht_CAN4_7DD6_Tx.Data[0]	:=	Brusa1_Rx.ActLim_Rx.au8_Data[0];
ht_CAN4_7DD6_Tx.Data[1]	:=	Brusa1_Rx.ActLim_Rx.au8_Data[1];
ht_CAN4_7DD6_Tx.Data[2]	:=	Brusa1_Rx.ActLim_Rx.au8_Data[2];
ht_CAN4_7DD6_Tx.Data[3]	:=	Brusa1_Rx.ActLim_Rx.au8_Data[3];
ht_CAN4_7DD6_Tx.Data[4]	:=	Brusa1_Rx.ActLim_Rx.au8_Data[4];
ht_CAN4_7DD6_Tx.Data[5]	:=	Brusa1_Rx.ActLim_Rx.au8_Data[5];
ht_CAN4_7DD6_Tx.Data[6]	:=	Brusa1_Rx.ActLim_Rx.au8_Data[6];
ht_CAN4_7DD6_Tx.Data[7]	:=	Brusa1_Rx.ActLim_Rx.au8_Data[7];
ht_CAN4_7DD6_Tx.Len		:=	8;

ht_CAN4_7DD8_Tx.ID		:=	16#187008DD OR EPEC_CANVXD.MASK_29BIT;
ht_CAN4_7DD8_Tx.Data[0]	:=	Brusa1_Rx.ActPlug_Rx.au8_Data[0];
ht_CAN4_7DD8_Tx.Data[1]	:=	Brusa1_Rx.ActPlug_Rx.au8_Data[1];
ht_CAN4_7DD8_Tx.Data[2]	:=	Brusa1_Rx.ActPlug_Rx.au8_Data[2];
ht_CAN4_7DD8_Tx.Data[3]	:=	Brusa1_Rx.ActPlug_Rx.au8_Data[3];
ht_CAN4_7DD8_Tx.Data[4]	:=	Brusa1_Rx.ActPlug_Rx.au8_Data[4];
ht_CAN4_7DD8_Tx.Data[5]	:=	Brusa1_Rx.ActPlug_Rx.au8_Data[5];
ht_CAN4_7DD8_Tx.Data[6]	:=	Brusa1_Rx.ActPlug_Rx.au8_Data[6];
ht_CAN4_7DD8_Tx.Data[7]	:=	Brusa1_Rx.ActPlug_Rx.au8_Data[7];
ht_CAN4_7DD8_Tx.Len		:=	8;

ht_CAN4_7DDA_Tx.ID		:=	16#18700ADD OR EPEC_CANVXD.MASK_29BIT;
ht_CAN4_7DDA_Tx.Data[0]	:=	Brusa1_Tx.DenLim_Tx.Data[0];
ht_CAN4_7DDA_Tx.Data[1]	:=	Brusa1_Tx.DenLim_Tx.Data[1];
ht_CAN4_7DDA_Tx.Data[2]	:=	Brusa1_Tx.DenLim_Tx.Data[2];
ht_CAN4_7DDA_Tx.Data[3]	:=	Brusa1_Tx.DenLim_Tx.Data[3];
ht_CAN4_7DDA_Tx.Data[4]	:=	Brusa1_Tx.DenLim_Tx.Data[4];
ht_CAN4_7DDA_Tx.Data[5]	:=	Brusa1_Tx.DenLim_Tx.Data[5];
ht_CAN4_7DDA_Tx.Data[6]	:=	Brusa1_Tx.DenLim_Tx.Data[6];
ht_CAN4_7DDA_Tx.Data[7]	:=	Brusa1_Tx.DenLim_Tx.Data[7];
ht_CAN4_7DDA_Tx.Len		:=	8;


//Slave Brusa
ht_CAN4_7DD1_Tx.ID		:=	16#187001DD OR EPEC_CANVXD.MASK_29BIT;
ht_CAN4_7DD1_Tx.Data[0]	:=	Brusa2_Rx.ActAC_Rx.au8_Data[0];
ht_CAN4_7DD1_Tx.Data[1]	:=	Brusa2_Rx.ActAC_Rx.au8_Data[1];
ht_CAN4_7DD1_Tx.Data[2]	:=	Brusa2_Rx.ActAC_Rx.au8_Data[2];
ht_CAN4_7DD1_Tx.Data[3]	:=	Brusa2_Rx.ActAC_Rx.au8_Data[3];
ht_CAN4_7DD1_Tx.Data[4]	:=	Brusa2_Rx.ActAC_Rx.au8_Data[4];
ht_CAN4_7DD1_Tx.Data[5]	:=	Brusa2_Rx.ActAC_Rx.au8_Data[5];
ht_CAN4_7DD1_Tx.Data[6]	:=	Brusa2_Rx.ActAC_Rx.au8_Data[6];
ht_CAN4_7DD1_Tx.Data[7]	:=	Brusa2_Rx.ActAC_Rx.au8_Data[7];
ht_CAN4_7DD1_Tx.Len		:=	8;

ht_CAN4_7DD3_Tx.ID		:=	16#187003DD OR EPEC_CANVXD.MASK_29BIT;
ht_CAN4_7DD3_Tx.Data[0]	:=	Brusa2_Rx.NLG2_ActErr_Rx.au8_Data[0];
ht_CAN4_7DD3_Tx.Data[1]	:=	Brusa2_Rx.NLG2_ActErr_Rx.au8_Data[1];
ht_CAN4_7DD3_Tx.Data[2]	:=	Brusa2_Rx.NLG2_ActErr_Rx.au8_Data[2];
ht_CAN4_7DD3_Tx.Data[3]	:=	Brusa2_Rx.NLG2_ActErr_Rx.au8_Data[3];
ht_CAN4_7DD3_Tx.Data[4]	:=	Brusa2_Rx.NLG2_ActErr_Rx.au8_Data[4];
ht_CAN4_7DD3_Tx.Data[5]	:=	Brusa2_Rx.NLG2_ActErr_Rx.au8_Data[5];
ht_CAN4_7DD3_Tx.Data[6]	:=	Brusa2_Rx.NLG2_ActErr_Rx.au8_Data[6];
ht_CAN4_7DD3_Tx.Data[7]	:=	Brusa2_Rx.NLG2_ActErr_Rx.au8_Data[7];
ht_CAN4_7DD3_Tx.Len		:=	8;

ht_CAN4_7DD5_Tx.ID		:=	16#187005DD OR EPEC_CANVXD.MASK_29BIT;
ht_CAN4_7DD5_Tx.Data[0]	:=	Brusa2_Rx.NLG2_ActInt_Rx.au8_Data[0];
ht_CAN4_7DD5_Tx.Data[1]	:=	Brusa2_Rx.NLG2_ActInt_Rx.au8_Data[1];
ht_CAN4_7DD5_Tx.Data[2]	:=	Brusa2_Rx.NLG2_ActInt_Rx.au8_Data[2];
ht_CAN4_7DD5_Tx.Data[3]	:=	Brusa2_Rx.NLG2_ActInt_Rx.au8_Data[3];
ht_CAN4_7DD5_Tx.Data[4]	:=	Brusa2_Rx.NLG2_ActInt_Rx.au8_Data[4];
ht_CAN4_7DD5_Tx.Data[5]	:=	Brusa2_Rx.NLG2_ActInt_Rx.au8_Data[5];
ht_CAN4_7DD5_Tx.Data[6]	:=	Brusa2_Rx.NLG2_ActInt_Rx.au8_Data[6];
ht_CAN4_7DD5_Tx.Data[7]	:=	Brusa2_Rx.NLG2_ActInt_Rx.au8_Data[7];
ht_CAN4_7DD5_Tx.Len		:=	8;

ht_CAN4_7DD7_Tx.ID		:=	16#187007DD OR EPEC_CANVXD.MASK_29BIT;
ht_CAN4_7DD7_Tx.Data[0]	:=	Brusa2_Rx.NLG2_ActLim_Rx.au8_Data[0];
ht_CAN4_7DD7_Tx.Data[1]	:=	Brusa2_Rx.NLG2_ActLim_Rx.au8_Data[1];
ht_CAN4_7DD7_Tx.Data[2]	:=	Brusa2_Rx.NLG2_ActLim_Rx.au8_Data[2];
ht_CAN4_7DD7_Tx.Data[3]	:=	Brusa2_Rx.NLG2_ActLim_Rx.au8_Data[3];
ht_CAN4_7DD7_Tx.Data[4]	:=	Brusa2_Rx.NLG2_ActLim_Rx.au8_Data[4];
ht_CAN4_7DD7_Tx.Data[5]	:=	Brusa2_Rx.NLG2_ActLim_Rx.au8_Data[5];
ht_CAN4_7DD7_Tx.Data[6]	:=	Brusa2_Rx.NLG2_ActLim_Rx.au8_Data[6];
ht_CAN4_7DD7_Tx.Data[7]	:=	Brusa2_Rx.NLG2_ActLim_Rx.au8_Data[7];
ht_CAN4_7DD7_Tx.Len		:=	8;

ht_CAN4_7DD9_Tx.ID		:=	16#187009DD OR EPEC_CANVXD.MASK_29BIT;
ht_CAN4_7DD9_Tx.Data[0]	:=	Brusa2_Rx.NLG2_ActPlug_Rx.au8_Data[0];
ht_CAN4_7DD9_Tx.Data[1]	:=	Brusa2_Rx.NLG2_ActPlug_Rx.au8_Data[1];
ht_CAN4_7DD9_Tx.Data[2]	:=	Brusa2_Rx.NLG2_ActPlug_Rx.au8_Data[2];
ht_CAN4_7DD9_Tx.Data[3]	:=	Brusa2_Rx.NLG2_ActPlug_Rx.au8_Data[3];
ht_CAN4_7DD9_Tx.Data[4]	:=	Brusa2_Rx.NLG2_ActPlug_Rx.au8_Data[4];
ht_CAN4_7DD9_Tx.Data[5]	:=	Brusa2_Rx.NLG2_ActPlug_Rx.au8_Data[5];
ht_CAN4_7DD9_Tx.Data[6]	:=	Brusa2_Rx.NLG2_ActPlug_Rx.au8_Data[6];
ht_CAN4_7DD9_Tx.Data[7]	:=	Brusa2_Rx.NLG2_ActPlug_Rx.au8_Data[7];
ht_CAN4_7DD9_Tx.Len		:=	8;

ht_CAN4_7DDB_Tx.ID		:=	16#18700BDD OR EPEC_CANVXD.MASK_29BIT;
ht_CAN4_7DDB_Tx.Data[0]	:=	Brusa2_Tx.DenLim_Tx.Data[0];
ht_CAN4_7DDB_Tx.Data[1]	:=	Brusa2_Tx.DenLim_Tx.Data[1];
ht_CAN4_7DDB_Tx.Data[2]	:=	Brusa2_Tx.DenLim_Tx.Data[2];
ht_CAN4_7DDB_Tx.Data[3]	:=	Brusa2_Tx.DenLim_Tx.Data[3];
ht_CAN4_7DDB_Tx.Data[4]	:=	Brusa2_Tx.DenLim_Tx.Data[4];
ht_CAN4_7DDB_Tx.Data[5]	:=	Brusa2_Tx.DenLim_Tx.Data[5];
ht_CAN4_7DDB_Tx.Data[6]	:=	Brusa2_Tx.DenLim_Tx.Data[6];
ht_CAN4_7DDB_Tx.Data[7]	:=	Brusa2_Tx.DenLim_Tx.Data[7];
ht_CAN4_7DDB_Tx.Len		:=	8;



Tx_Timer(IN := NOT(Tx_Timer.Q), PT := T#100MS);
IF (Tx_Timer.Q = TRUE) THEN
	G_CAN4_Channel.SendMessage(i_pMSG:=ADR(ht_CAN4_7DD0_Tx));
	G_CAN4_Channel.SendMessage(i_pMSG:=ADR(ht_CAN4_7DD1_Tx));
	G_CAN4_Channel.SendMessage(i_pMSG:=ADR(ht_CAN4_7DD2_Tx));
	G_CAN4_Channel.SendMessage(i_pMSG:=ADR(ht_CAN4_7DD3_Tx));
	G_CAN4_Channel.SendMessage(i_pMSG:=ADR(ht_CAN4_7DD4_Tx));
	G_CAN4_Channel.SendMessage(i_pMSG:=ADR(ht_CAN4_7DD5_Tx));
	G_CAN4_Channel.SendMessage(i_pMSG:=ADR(ht_CAN4_7DD6_Tx));
	G_CAN4_Channel.SendMessage(i_pMSG:=ADR(ht_CAN4_7DD7_Tx));
	G_CAN4_Channel.SendMessage(i_pMSG:=ADR(ht_CAN4_7DD8_Tx));
	G_CAN4_Channel.SendMessage(i_pMSG:=ADR(ht_CAN4_7DD9_Tx));
	G_CAN4_Channel.SendMessage(i_pMSG:=ADR(ht_CAN4_7DDA_Tx));
	G_CAN4_Channel.SendMessage(i_pMSG:=ADR(ht_CAN4_7DDB_Tx));
END_IF

END_PROGRAM

// Application/UserCode/CAN1/CAN1_Tx
PROGRAM CAN1_Tx
VAR
	ht_EEC1_Tx	:	EPEC_CANVXD.Msg;
	ht_EEC2_Tx	:	EPEC_CANVXD.Msg;
	ht_EEC3_Tx	:	EPEC_CANVXD.Msg;
	ht_CCSS_Tx	:	EPEC_CANVXD.Msg;
	ht_Allison_Override_Tx: EPEC_CANVXD.Msg;
	ht_SOCDash_Tx	:	EPEC_CANVXD.Msg;
	ht_TemperatureDash	:	EPEC_CANVXD.Msg;
	ht_TransmissionWarning_Bob_Tx	:	EPEC_CANVXD.Msg;
	
	hton_MessageSend_Timer	:	TON;
	hton_MessageSend1sec_Timer	:	TON;
	
	ht_Allison_ETC7_Tx	:	EPEC_CANVXD.Msg;
	ht_Allison_ProbA_Tx	:	EPEC_CANVXD.Msg;
	
	ht_SpeedDisplay_Tx	:	EPEC_CANVXD.Msg;
	ht_ExhaustAftertreatment_Tx	:	EPEC_CANVXD.Msg;
	
	ht_RearSteerActive_Tx	:	EPEC_CANVXD.Msg;
	ht_TracStabReport_Tx	:	EPEC_CANVXD.Msg;
	
	(*ht_Test	:	EPEC_CANVXD.Msg;
	hu8_TestCounter	:	USINT;
	hu8_TestChecksum	:	USINT;
	hton_TestTimer	:	TON;*)
	
	hu8_EEC1_Byte0	:	USINT;
	hu8_EEC2_Byte0	:	USINT;
	hu8_EEC2_Byte5	:	USINT;
	hu8_EEC3_Byte7	:	USINT;
END_VAR


CAN1_TxConversion();

(*Combining transmit variables into bytes*)
hu8_EEC1_Byte0	:=	(gu8_ENG_EngineTorqueMode AND 2#00001111) +
					(SHL(gu8_ENG_ActlEngPrcntTorqueHghResolution_Tx, 4) AND 2#11110000);
hu8_EEC2_Byte0	:=	(gu8_ENG_AccelPedal1LowIdleSwitch AND 2#00000011) +
					(SHL(gu8_ENG_AccelPedalKickdownSwitch, 2) AND 2#00001100) +
					(SHL(gu8_ENG_RoadSpeedLimitStatus, 4) AND 2#00110000) +
					(SHL(gu8_ENG_AccelPedal2LowIdleSwitch, 6) AND 2#11000000);
hu8_EEC2_Byte5	:=	(gu8_ENG_VehicleAccelRateLimitStatus AND 2#00000011) +
					(SHL(gu8_ENG_MomentaryEngMaxPowEnableFeedback, 2) AND 2#00001100) +
					(SHL(gu8_ENG_DPFThermalManagementActive, 4) AND 2#00110000) +
					(SHL(gu8_ENG_SCRThermalManagementActive, 6) AND 2#11000000);
hu8_EEC3_Byte7	:=	(gu8_ENG_Aftertreatment1IntakeDewPoint AND 2#00000011) +
					(SHL(gu8_ENG_Aftertreatment1ExhaustDewPoint, 2) AND 2#00001100) +
					(SHL(gu8_ENG_Aftertreatment2IntakeDewPoint, 4) AND 2#00110000) +
					(SHL(gu8_ENG_Aftertreatment2ExhaustDewPoint, 6) AND 2#11000000);

{region "KB"}
(*Set the transmit data for the messages to be sent*)
ht_EEC1_Tx.ID		:=	16#0CF00400  OR EPEC_CANVXD.MASK_29BIT;
ht_EEC1_Tx.Data[0]	:=	hu8_EEC1_Byte0;
ht_EEC1_Tx.Data[1]	:=	gu8_ENG_DriversDemandEnginePercentTorque;
ht_EEC1_Tx.Data[2]	:=	gu8_ENG_ActualEnginePercentTorque;
ht_EEC1_Tx.Data[3]	:=	UINT_TO_USINT(gu16_ENG_EngineSpeed_Tx);
ht_EEC1_Tx.Data[4]	:=	UINT_TO_USINT(SHR(gu16_ENG_EngineSpeed_Tx, 8));
ht_EEC1_Tx.Data[5]	:=	gu8_ENG_SrcAddrOfCtrllingDevForEngCtrl;
ht_EEC1_Tx.Data[6]	:=	gu8_ENG_EngineStarterMode;
ht_EEC1_Tx.Data[7]	:=	gu8_ENG_EngineDemandPercentTorque;
ht_EEC1_Tx.Len		:=	8;

ht_EEC2_Tx.ID		:=	16#0CF00300 OR EPEC_CANVXD.MASK_29BIT;
ht_EEC2_Tx.Data[0]	:=	hu8_EEC2_Byte0;
ht_EEC2_Tx.Data[1]	:=	gu8_ENG_AccelPedalPosition_Tx;
ht_EEC2_Tx.Data[2]	:=	gu8_ENG_EnginePercLoadCurrentSpeed;
ht_EEC2_Tx.Data[3]	:=	gu8_ENG_RemoteAccelPedalPosition_Tx;
ht_EEC2_Tx.Data[4]	:=	gu8_ENG_AccelPedalPosition2_Tx;
ht_EEC2_Tx.Data[5]	:=	hu8_EEC2_Byte5;
ht_EEC2_Tx.Data[6]	:=	gu8_ENG_ActualMaxAvailableEngPercTorque_Tx;
ht_EEC2_Tx.Data[7]	:=	gu8_ENG_EstimatedPumpingPercentTorque;
ht_EEC2_Tx.Len		:=	8;

ht_EEC3_Tx.ID		:=	16#18FEDF00 OR EPEC_CANVXD.MASK_29BIT;
ht_EEC3_Tx.Data[0]	:=	gu8_ENG_NominalFrictionPercTorque;
ht_EEC3_Tx.Data[1]	:=	UINT_TO_USINT(gu16_ENG_EngDesiredOperatingSpeed_Tx);
ht_EEC3_Tx.Data[2]	:=	UINT_TO_USINT(SHR(gu16_ENG_EngDesiredOperatingSpeed_Tx, 8));
ht_EEC3_Tx.Data[3]	:=	gu8_ENG_EngDesiredOperatingSpeedAsymAdjust;
ht_EEC3_Tx.Data[4]	:=	gu8_ENG_EstEngParasiticLossPercTorque;
ht_EEC3_Tx.Data[5]	:=	UINT_TO_USINT(gu16_ENG_Aftertreatment1ExhaustGasMassFlow_Tx);
ht_EEC3_Tx.Data[6]	:=	UINT_TO_USINT(SHR(gu16_ENG_Aftertreatment1ExhaustGasMassFlow_Tx, 8));
ht_EEC3_Tx.Data[7]	:=	hu8_EEC3_Byte7;
ht_EEC3_Tx.Len		:=	8;

ht_CCSS_Tx.ID		:=	16#18FEED00 OR EPEC_CANVXD.MASK_29BIT;
ht_CCSS_Tx.Data[0]	:=	gu8_ENG_MaxVehicleSpeedLimit;
ht_CCSS_Tx.Data[1]	:=	gu8_ENG_CruiseControlHighSetSpeedLimit;
ht_CCSS_Tx.Data[2]	:=	gu8_ENG_CruiseControlLowSetSpeedLimit;
ht_CCSS_Tx.Data[3]	:=	0;
ht_CCSS_Tx.Data[4]	:=	0;
ht_CCSS_Tx.Data[5]	:=	0;
ht_CCSS_Tx.Data[6]	:=	0;
ht_CCSS_Tx.Data[7]	:=	0;
ht_CCSS_Tx.Len		:=	8;
	 
(*Allison Selector Return*)
ht_Allison_ETC7_Tx.ID		:=	16#18FE4AD3 OR EPEC_CANVXD.MASK_29BIT;
ht_Allison_ETC7_Tx.Data[0]	:=	16#03;
ht_Allison_ETC7_Tx.Data[1]	:=	gu8_ETC7_TransmissionEngaged_Tx;
ht_Allison_ETC7_Tx.Data[2]	:=	16#4F;
ht_Allison_ETC7_Tx.Data[3]	:=	16#E0;
ht_Allison_ETC7_Tx.Data[4]	:=	16#FF;
ht_Allison_ETC7_Tx.Data[5]	:=	16#F3;
ht_Allison_ETC7_Tx.Data[6]	:=	16#FF;
ht_Allison_ETC7_Tx.Data[7]	:=	16#FF;
ht_Allison_ETC7_Tx.Len		:=	8;

ht_Allison_ProbA_Tx.ID		:=	16#18EF0503 OR EPEC_CANVXD.MASK_29BIT;
ht_Allison_ProbA_Tx.Data[0]	:=	16#0A;
ht_Allison_ProbA_Tx.Data[1]	:=	16#FC;
ht_Allison_ProbA_Tx.Data[2]	:=	16#00;
ht_Allison_ProbA_Tx.Data[3]	:=	16#01;
ht_Allison_ProbA_Tx.Data[4]	:=	16#23;
ht_Allison_ProbA_Tx.Data[5]	:=	16#01;
ht_Allison_ProbA_Tx.Data[6]	:=	gu8_ProbA_GearSelected_Tx;
ht_Allison_ProbA_Tx.Data[7]	:=	gu8_ProbA_GearSelected_Tx;
ht_Allison_ProbA_Tx.Len		:=	8;

ht_SpeedDisplay_Tx.ID		:=	16#18FF82C4 OR EPEC_CANVXD.MASK_29BIT;
ht_SpeedDisplay_Tx.Data[0]	:=	REAL_TO_USINT(gr_VehicleSpeed_kmph);
ht_SpeedDisplay_Tx.Data[1]	:=	0;
ht_SpeedDisplay_Tx.Data[2]	:=	0;
ht_SpeedDisplay_Tx.Data[3]	:=	0;
ht_SpeedDisplay_Tx.Data[4]	:=	0;
ht_SpeedDisplay_Tx.Data[5]	:=	0;
ht_SpeedDisplay_Tx.Data[6]	:=	0;
ht_SpeedDisplay_Tx.Data[7]	:=	0;
ht_SpeedDisplay_Tx.Len		:=	8;
	 
ht_Allison_Override_Tx.ID			:= 16#18FF0400 OR EPEC_CANVXD.MASK_29BIT;
ht_Allison_Override_Tx.Data[1]		:=	0;
ht_Allison_Override_Tx.Data[2]		:=	0;
ht_Allison_Override_Tx.Data[3]		:=	0;
ht_Allison_Override_Tx.Data[4].0	:=	gq_Gear_Neutral;
ht_Allison_Override_Tx.Data[4].1	:=	gq_Gear_Drive;
ht_Allison_Override_Tx.Data[4].2	:=	gq_Gear_Reverse;
ht_Allison_Override_Tx.Data[5]		:=	0;
ht_Allison_Override_Tx.Data[6]		:=	0;
ht_Allison_Override_Tx.Data[7]		:=	0;
ht_Allison_Override_Tx.Len			:=	8;

ht_SOCDash_Tx.ID			:=	16#18FF013D OR EPEC_CANVXD.MASK_29BIT;
ht_SOCDash_Tx.Data[0]		:=	WORD_TO_BYTE (Dennis_Regen.RegenCounterValue);
ht_SOCDash_Tx.Data[1]		:=	0;
ht_SOCDash_Tx.Data[2]		:=	0;
ht_SOCDash_Tx.Data[3]		:=	0;
ht_SOCDash_Tx.Data[4]		:=	REAL_TO_USINT(gu8_BMS_SOC * 2.4); (* What is the scale about?? Luke Matt *)
ht_SOCDash_Tx.Data[5]		:=	16#3A;
ht_SOCDash_Tx.Data[6]		:=	0;
ht_SOCDash_Tx.Data[7]		:=	0;
ht_SOCDash_Tx.Len			:=	8;
	 
ht_TemperatureDash.ID		:=	16#0 OR EPEC_CANVXD.MASK_29BIT;
ht_TemperatureDash.Data[0]	:=	0;
ht_TemperatureDash.Data[1]	:=	0;
ht_TemperatureDash.Data[2]	:=	0;
ht_TemperatureDash.Data[3]	:=	0;
ht_TemperatureDash.Data[4]	:=	0;
ht_TemperatureDash.Data[5]	:=	0;
ht_TemperatureDash.Data[6]	:=	0;
ht_TemperatureDash.Data[7]	:=	0;
ht_TemperatureDash.Len		:=	8;

ht_ExhaustAftertreatment_Tx.ID	:=	16#18FF043D OR EPEC_CANVXD.MASK_29BIT;
ht_ExhaustAftertreatment_Tx.Data[0]	:=	0;
ht_ExhaustAftertreatment_Tx.Data[1]	:=	0;
ht_ExhaustAftertreatment_Tx.Data[2]	:=	0;  
ht_ExhaustAftertreatment_Tx.Data[3]	:=	0;  
ht_ExhaustAftertreatment_Tx.Data[4]	:=	0;  
ht_ExhaustAftertreatment_Tx.Data[5]	:=	0;  
ht_ExhaustAftertreatment_Tx.Data[6]	:=	0;  
ht_ExhaustAftertreatment_Tx.Data[7]	:=	0;
ht_ExhaustAftertreatment_Tx.Len		:=	8;  
	
	 
ht_TracStabReport_Tx.ID				:=	16#18FF400B OR EPEC_CANVXD.MASK_29BIT;
ht_TracStabReport_Tx.Data[0]		:=	gu8_TractionLoss;
ht_TracStabReport_Tx.Data[1]		:=	gu8_StabilityLoss;
ht_TracStabReport_Tx.Data[2].0		:=	Driveability.SecretTractionOff;
ht_TracStabReport_Tx.Data[3]		:=	0;
ht_TracStabReport_Tx.Data[4]		:=	0;
ht_TracStabReport_Tx.Data[5]		:=	0;
ht_TracStabReport_Tx.Data[6]		:=	0;
ht_TracStabReport_Tx.Data[7]		:=	0;
ht_TracStabReport_Tx.Len			:=	8;
	 
ht_TransmissionWarning_Bob_Tx.ID		:=	16#10FF0003 OR EPEC_CANVXD.MASK_29BIT;
ht_TransmissionWarning_Bob_Tx.Data[0]	:=	16#41;
ht_TransmissionWarning_Bob_Tx.Data[1]	:=	16#48;
ht_TransmissionWarning_Bob_Tx.Data[2]	:=	0;
ht_TransmissionWarning_Bob_Tx.Data[3]	:=	0;
ht_TransmissionWarning_Bob_Tx.Data[4]	:=	0;
ht_TransmissionWarning_Bob_Tx.Data[5]	:=	0;
ht_TransmissionWarning_Bob_Tx.Data[6]	:=	0;
ht_TransmissionWarning_Bob_Tx.Data[7]	:=	0;
ht_TransmissionWarning_Bob_Tx.Len		:=	8;
		  
	 
(*ht_RearSteerActive_Tx.ID	:=	16#18FF0401 OR EPEC_CANVXD.MASK_29BIT;
ht_RearSteerActive_Tx.Data[0]		:=	16#95;
ht_RearSteerActive_Tx.Data[1]		:=	16#FF;
ht_RearSteerActive_Tx.Data[2]		:=	16#FF;
ht_RearSteerActive_Tx.Data[3]		:=	16#41;
ht_RearSteerActive_Tx.Data[4]		:=	16#FA;
ht_RearSteerActive_Tx.Data[5]		:=	16#00;
ht_RearSteerActive_Tx.Data[6]		:=	16#0F;
ht_RearSteerActive_Tx.Data[7]		:=	16#C3;
ht_RearSteerActive_Tx.Len			:=	8;

ht_RearSteerActive_Tx.ID	:=	16#18FF0801 OR EPEC_CANVXD.MASK_29BIT;
ht_RearSteerActive_Tx.Data[0]		:=	16#FF;
ht_RearSteerActive_Tx.Data[1]		:=	16#FF;	
ht_RearSteerActive_Tx.Data[2]		:=	16#FA;	
ht_RearSteerActive_Tx.Data[3]		:=	16#FA;	
ht_RearSteerActive_Tx.Data[4]		:=	16#00;	
ht_RearSteerActive_Tx.Data[5]		:=	16#00;	
ht_RearSteerActive_Tx.Data[6]		:=	16#00;	
ht_RearSteerActive_Tx.Data[7]		:=	16#00;	
ht_RearSteerActive_Tx.Len			:=	8;*)

(*
ht_Test.ID			:=	16#0CFF0203 OR EPEC_CANVXD.MASK_29BIT;
ht_Test.Data[0]		:=	16#80;
ht_Test.Data[1]		:=	16#7D;
ht_Test.Data[2]		:=	16#FF;
ht_Test.Data[3]		:=	16#FF;
ht_Test.Data[4]		:=	16#FF;
ht_Test.Data[5]		:=	16#FF;
ht_Test.Data[6]		:=	(hu8_TestCounter * 16);
CASE (hu8_TestCounter) OF
	0: hu8_TestChecksum := 112;
	1: hu8_TestChecksum := 66;
	2: hu8_TestChecksum := 20;
	3: hu8_TestChecksum := 38;
	4: hu8_TestChecksum := 184;
	5: hu8_TestChecksum := 138;
	6: hu8_TestChecksum := 220;
	7: hu8_TestChecksum := 238;
	8: hu8_TestChecksum := 123;
	9: hu8_TestChecksum := 73;
	10: hu8_TestChecksum := 31;
	11: hu8_TestChecksum := 45;
	12: hu8_TestChecksum := 179;
	13: hu8_TestChecksum := 129;
	14: hu8_TestChecksum := 215;
	15:	hu8_TestChecksum := 229;
END_CASE
ht_Test.Data[7]		:=	hu8_TestChecksum;
ht_Test.Len			:=	8;*)
	 


			   
{endregion}
	 
{region "Send Messages"}
(*Transmit these messages*)
hton_MessageSend_Timer(IN := NOT(hton_MessageSend_Timer.Q), PT := T#60MS);
IF (hton_MessageSend_Timer.Q = TRUE) THEN
	G_CAN1_Channel.SendMessage(i_pMSG:=ADR(ht_EEC1_Tx));
	G_CAN1_Channel.SendMessage(i_pMSG:=ADR(ht_EEC2_Tx));
	G_CAN1_Channel.SendMessage(i_pMSG:=ADR(ht_EEC3_Tx));
	G_CAN1_Channel.SendMessage(i_pMSG:=ADR(ht_CCSS_Tx));
		 
	G_CAN1_Channel.SendMessage(i_pMSG:=ADR(ht_Allison_ETC7_Tx));
	G_CAN1_Channel.SendMessage(i_pMSG:=ADR(ht_Allison_ProbA_Tx));
		 
	G_CAN1_Channel.SendMessage(i_pMSG:=ADR(ht_ExhaustAftertreatment_Tx));
		 
	G_CAN1_Channel.SendMessage(i_pMSG:=ADR(ht_TracStabReport_Tx));
	G_CAN1_Channel.SendMessage(i_pMSG:=ADR(ht_TransmissionWarning_Bob_Tx));  
END_IF
hton_MessageSend1sec_Timer(IN := NOT(hton_MessageSend1sec_Timer.Q), PT := T#1000MS);
IF (hton_MessageSend1sec_Timer.Q = TRUE) THEN
	G_CAN1_Channel.SendMessage(i_pMSG:=ADR(ht_SOCDash_Tx));
	G_CAN1_Channel.SendMessage(i_pMSG:=ADR(ht_RearSteerActive_Tx));
END_IF

IF (hton_MessageSend_Timer.Q = TRUE AND gq_Allison_Pad_Override = TRUE) THEN
	G_CAN1_Channel.SendMessage(i_pMSG:=ADR(ht_Allison_Override_Tx));
END_IF	 
		  
(*hton_TestTimer(IN := NOT(hton_TestTimer.Q), PT := T#50MS);
IF (hton_TestTimer.Q = TRUE) THEN
	(*hu8_TestCounter := hu8_TestCounter + 1;
	IF (hu8_TestCounter > 15) THEN
		hu8_TestCounter := 0;
	END_IF*)
	G_CAN1_Channel.SendMessage(i_pMSG:=ADR(ht_Test)); 
END_IF*)
{endregion}

END_PROGRAM

// Application/UserCode/CAN1/CAN1_TxConversion
PROGRAM CAN1_TxConversion
VAR
	RPM_READY_GAUGE	:	UINT	:=	2816; (*Minimum value needed so that rear steer will activate*)
END_VAR
VAR CONSTANT
	DRIVEENGAGED	:	USINT	:=	3;
	DRIVEDISENGAGED	:	USINT	:=	19;
	
	GEAR_DRIVE		:	USINT	:=	68;
	GEAR_REVERSE	:	USINT	:=	82;
	GEAR_NEUTRAL	:	USINT	:=	78;
	
	MCU_OPERATIONAL		:	USINT	:=	4;
END_VAR


(*Tx preconversion*)
(*EEC1*)
gr_ENG_ActlEngPrcntTorqueHghResolution		:=	0;
gr_ENG_EngineSpeed							:=	LIMIT(500, (ABS(gr_BMS_BatteryVoltage * gs16_BMS_BatteryCurrent) + 1500), 2700) (*Batt power + 1500 Lim(500->2700) * CF*);
(*EEC2*)
gr_ENG_AccelPedalPosition1					:=	gr_AccelPedal_Perc;
gr_ENG_RemoteAccelPedalPosition				:=	0;
gr_ENG_AccelPedalPosition2					:=	0;
gr_ENG_ActualMaxAvailableEngPercTorque		:=	0;
(*EEC3*)
gr_ENG_EngDesiredOperatingSpeed				:=	0;
gr_ENG_AfterTreatment1ExhaustGasMassFlow	:=	0;

(*Need to swap all the signed intergers over to unsigned so it can be processed correctly*)

(*EEC1*) (*0C FF 7D DisplayRPM Display RPM 00 FF 7D*)
gu8_ENG_EngineTorqueMode					:=	12; (*Need to define why currently no enumeration for this*)
gu8_ENG_ActlEngPrcntTorqueHghResolution_Tx	:=	REAL_TO_USINT(gr_ENG_ActlEngPrcntTorqueHghResolution);
gu8_ENG_DriversDemandEnginePercentTorque	:=	16#FF; (*Need to define this, no current enumeration*)
gu8_ENG_ActualEnginePercentTorque			:=	0;
gu16_ENG_EngineSpeed_Tx						:=	REAL_TO_UINT(gr_ENG_EngineSpeed / 0.125);
gu8_ENG_SrcAddrOfCtrllingDevForEngCtrl			:=	0;
gu8_ENG_EngineStarterMode						:=	0;
gu8_ENG_EngineDemandPercentTorque				:=	0;
(*EEC2*) (*FF FF 00 FF FF 0F 00 00*)
gu8_ENG_AccelPedal1LowIdleSwitch			:=	0;
gu8_ENG_AccelPedalKickdownSwitch			:=	0;
gu8_ENG_RoadSpeedLimitStatus				:=	0;
gu8_ENG_AccelPedal2LowIdleSwitch			:=	0;
gu8_ENG_AccelPedalPosition_Tx				:=	0;
gu8_ENG_EnginePercLoadCurrentSpeed			:=	0;
gu8_ENG_RemoteAccelPedalPosition_Tx			:=	0;
gu8_ENG_AccelPedalPosition2_Tx				:=	0;
gu8_ENG_VehicleAccelRateLimitStatus			:=	0;
gu8_ENG_MomentaryEngMaxPowEnableFeedback	:=	0;
gu8_ENG_DPFThermalManagementActive			:=	0;
gu8_ENG_SCRThermalManagementActive			:=	0;
gu8_ENG_ActualMaxAvailableEngPercTorque_Tx	:=	0;
gu8_ENG_EstimatedPumpingPercentTorque		:=	0;
(*EEC3*) (*86 40 1F 7D 7D FF FF FF*)
gu8_ENG_NominalFrictionPercTorque			:=	0;
gu16_ENG_EngDesiredOperatingSpeed_Tx		:=	0;
gu8_ENG_EngDesiredOperatingSpeedAsymAdjust	:=	0;
gu8_ENG_EstEngParasiticLossPercTorque		:=	0;
gu16_ENG_Aftertreatment1ExhaustGasMassFlow_Tx	:=	0;
gu8_ENG_Aftertreatment1IntakeDewPoint		:=	0;
gu8_ENG_Aftertreatment1ExhaustDewPoint		:=	0;
gu8_ENG_Aftertreatment2IntakeDewPoint		:=	0;
gu8_ENG_Aftertreatment2ExhaustDewPoint		:=	0;
(*CCSS*) (*FA 64 00 FF FF FF FF FF*)
gu8_ENG_MaxVehicleSpeedLimit				:=	0;
gu8_ENG_CruiseControlHighSetSpeedLimit		:=	0;
gu8_ENG_CruiseControlLowSetSpeedLimit		:=	0;
(******************************************************************************************************************************************)
(******************************************************************************************************************************************)
(*Values to send to the Allison to get it to display*)
IF (gq_Gear_Drive = TRUE OR	gq_Gear_DriveCrawl = TRUE OR gq_Gear_Reverse = TRUE OR gq_Gear_ReverseCrawl	= TRUE) THEN
	gu8_ETC7_TransmissionEngaged_Tx	:=	DRIVEENGAGED;
ELSE
	gu8_ETC7_TransmissionEngaged_Tx	:=	DRIVEDISENGAGED;
END_IF
IF (gq_Gear_Drive = TRUE OR	gq_Gear_DriveCrawl = TRUE) THEN
	gu8_ProbA_GearSelected_Tx	:=	GEAR_DRIVE;
ELSIF (gq_Gear_Reverse = TRUE OR gq_Gear_ReverseCrawl	= TRUE) THEN
	gu8_ProbA_GearSelected_Tx	:=	GEAR_REVERSE;
ELSE
	gu8_ProbA_GearSelected_Tx	:=	GEAR_NEUTRAL;
END_IF

IF (DO_q_DashboardDCDCStatus_DO = TRUE) THEN
	gu16_RPM_Display	:=	RPM_READY_GAUGE;
ELSE
	gu16_RPM_Display	:=	0;
END_IF


gu16_MCM02_EngineTorque_Tx	:=	REAL_TO_UINT(((LIMIT(-5000, gr_MCU_MotorTorqueEstimated, 5000) + 5000) / 0.2));
gu16_TCM03_ShaftSpeed_Tx	:=	REAL_TO_UINT(LIMIT(0, ABS(gr_MCU_MotorSpeed), 8000) / 0.16);

gu16_TCM2_OutputShaftSpeed	:=	REAL_TO_UINT(MIN(ABS(gr_MCU_MotorSpeed), 8000) / 0.16);
IF (gu8_MCU_State = MCU_OPERATIONAL) THEN
	gu8_TCM2_RotSens_Stat	:=	0;(*No Standstill*) (*1: Standstill, 2: Error*)
ELSE
	gu8_TCM2_RotSens_Stat	:=	3; (*SNA*)
END_IF
IF (gr_MCU_MotorSpeed >= 0) THEN
	gu8_TCM2_DrvDirec_Stat	:=	0; //FWD
ELSE
	gu8_TCM2_DrvDirec_Stat	:=	1; //BWD
END_IF

IF (gq_Gear_Drive = TRUE) THEN
	gu8_TCM8_Gear	:=	126;
	gu8_TCM8_DrvDirByGr_Stat	:=	2;
ELSIF (gq_Gear_Reverse = TRUE) THEN
	gu8_TCM8_Gear	:=	124;
	gu8_TCM8_DrvDirByGr_Stat	:=	0;
ELSE
	gu8_TCM8_Gear	:=	125;
	gu8_TCM8_DrvDirByGr_Stat	:=	1;
END_IF

gu16_TCM11_ActualGearRatio	:=	((gu16_GearRatio_PreCF / 1000) + 25) * 1000;

END_PROGRAM

// Application/UserCode/CAN4/Heater/Heater_Tx
PROGRAM Heater_Tx
VAR
	ht_CAN4_Heater_Tx	:	EPEC_CANVXD.Msg;
	ht_CAN4_OldHeater_Tx	:	EPEC_CANVXD.Msg;
	hq_OldHeater_Command: BOOL;
	hu8_Old_HeaterPerc	:	USINT;
	hu8_Old_HeaterTemp	:	USINT;
	
END_VAR


ht_CAN4_Heater_Tx.ID		:=	16#023;
ht_CAN4_Heater_Tx.Data[0]	:=	gu8_Heater_Perc;
ht_CAN4_Heater_Tx.Data[1]	:=	gu8_Heater_Temp_Tx;
ht_CAN4_Heater_Tx.Data[2]	:=	0;
ht_CAN4_Heater_Tx.Data[3]	:=	0;
ht_CAN4_Heater_Tx.Data[3].3	:=	gq_Heater_EnableBit;
ht_CAN4_Heater_Tx.Data[4]	:=	0;
ht_CAN4_Heater_Tx.Data[5]	:=	0;
ht_CAN4_Heater_Tx.Data[6]	:=	0;
ht_CAN4_Heater_Tx.Data[7]	:=	0;
ht_CAN4_Heater_Tx.Len		:=	8;

ht_CAN4_OldHeater_Tx.ID		:=	16#066;
ht_CAN4_OldHeater_Tx.Data[0]	:=	0;
ht_CAN4_OldHeater_Tx.Data[0].0	:=	gq_Heater_EnableBit;
ht_CAN4_OldHeater_Tx.Data[1]	:=	16#50;
ht_CAN4_OldHeater_Tx.Data[2]	:=	0;
ht_CAN4_OldHeater_Tx.Data[3]	:=	0;
ht_CAN4_OldHeater_Tx.Data[4]	:=	0;
ht_CAN4_OldHeater_Tx.Data[5]	:=	0;
ht_CAN4_OldHeater_Tx.Data[6]	:=	0;
ht_CAN4_OldHeater_Tx.Data[7]	:=	0;
ht_CAN4_OldHeater_Tx.Len		:=	8;


IF (gq_Heater_EnableBit <> hq_OldHeater_Command OR
	gu8_Heater_Perc <> hu8_Old_HeaterPerc OR ContactorControl.hq_BatteryDischargeMain_Rq OR
	gu8_Heater_Temp_Tx <> hu8_Old_HeaterTemp) THEN
	G_CAN4_Channel.SendMessage(i_pMSG:=ADR(ht_CAN4_Heater_Tx));
	G_CAN4_Channel.SendMessage(i_pMSG:=ADR(ht_CAN4_OldHeater_Tx));
END_IF

DO_q_HeaterOut_DI	:=	gq_HeaterPumpEnable;

hq_OldHeater_Command	:= gq_Heater_EnableBit;
hu8_Old_HeaterPerc		:=	gu8_Heater_Perc;
hu8_Old_HeaterTemp		:=	gu8_Heater_Temp_Tx;

END_PROGRAM

// Application/UserCode/CAN4/Heater/Heater_Rx
PROGRAM Heater_Rx
VAR
END_VAR

//Awaiting all the Data From the heater LDF
// All taken care of in HMI Code.
//So there MF>

END_PROGRAM

// Application/UserCode/ePTO/EPTO_Tx
PROGRAM EPTO_Tx
VAR
	MercCurrentGear1_Tx	:	EPEC_CANVXD.Msg;
	MercLHFWheelSpd_Tx	:	EPEC_CANVXD.Msg;
	MercCurrentGear2_Tx	:	EPEC_CANVXD.Msg;
	MercControlRPM_Tx	:	EPEC_CANVXD.Msg;
	ePTO_OilRq_Tx		:	EPEC_CANVXD.Msg;
	ePTO_Speed_47A_Tx	:	EPEC_CANVXD.Msg;
	ePTO_Torque_57A_Tx	:	EPEC_CANVXD.Msg;
	ePTO_NMT_Tx			:	EPEC_CANVXD.Msg;
	
	
	hton_MercePTO_TxTimer	:	TON;
END_VAR


{region "Data Allocation"}
(*Merc*)
MercCurrentGear1_Tx.ID := 16#18FE61EB OR EPEC_CANVXD.MASK_29BIT;
MercCurrentGear1_Tx.Data[0]	:=	0;
MercCurrentGear1_Tx.Data[1]	:=	gu8_CurrentGear2;
MercCurrentGear1_Tx.Data[2]	:=	0;
MercCurrentGear1_Tx.Data[3]	:=	0;
MercCurrentGear1_Tx.Data[4]	:=	0;
MercCurrentGear1_Tx.Data[5]	:=	0;
MercCurrentGear1_Tx.Data[6]	:=	0;
MercCurrentGear1_Tx.Data[7]	:=	0;
MercCurrentGear1_Tx.Len		:=	8;

MercLHFWheelSpd_Tx.ID := 16#0CFE5FEB OR EPEC_CANVXD.MASK_29BIT;
MercLHFWheelSpd_Tx.Data[0]	:=	0;
MercLHFWheelSpd_Tx.Data[1]	:=	0;
MercLHFWheelSpd_Tx.Data[2]	:=	0;
MercLHFWheelSpd_Tx.Data[3]	:=	03;
MercLHFWheelSpd_Tx.Data[4]	:=	20;
MercLHFWheelSpd_Tx.Data[5]	:=	0;
MercLHFWheelSpd_Tx.Data[6]	:=	UINT_TO_USINT(gu16_Bob_LeftFront_CAN);
MercLHFWheelSpd_Tx.Data[7]	:=	UINT_TO_USINT(SHR(gu16_Bob_LeftFront_CAN, 8));
MercLHFWheelSpd_Tx.Len		:=	8;

MercCurrentGear2_Tx.ID := 16#14FE80EB OR EPEC_CANVXD.MASK_29BIT;
MercCurrentGear2_Tx.Data[0]	:=	0;
MercCurrentGear2_Tx.Data[1]	:=	gu8_CurrentGear2;
MercCurrentGear2_Tx.Data[2]	:=	0;
MercCurrentGear2_Tx.Data[3]	:=	0;
MercCurrentGear2_Tx.Data[4]	:=	0;
MercCurrentGear2_Tx.Data[5]	:=	0;
MercCurrentGear2_Tx.Data[6]	:=	0;
MercCurrentGear2_Tx.Data[7]	:=	0;
MercCurrentGear2_Tx.Len		:=	8;

MercControlRPM_Tx.ID := 16#0CFE62C9 OR EPEC_CANVXD.MASK_29BIT;
MercControlRPM_Tx.Data[0]	:=	0;
MercControlRPM_Tx.Data[1]	:=	0;
MercControlRPM_Tx.Data[2]	:=	0;
MercControlRPM_Tx.Data[3]	:=	16#FA;
MercControlRPM_Tx.Data[4]	:=	0;
MercControlRPM_Tx.Data[5]	:=	0;
MercControlRPM_Tx.Data[6]	:=	0;
MercControlRPM_Tx.Data[7]	:=	0;
MercControlRPM_Tx.Len		:=	8;
	 
ePTO_OilRq_Tx.ID			:=	16#0CFF1355 OR EPEC_CANVXD.MASK_29BIT;
ePTO_OilRq_Tx.Data[0]		:=	0;
ePTO_OilRq_Tx.Data[1]		:=	0;
ePTO_OilRq_Tx.Data[2]		:=	0;
ePTO_OilRq_Tx.Data[3]		:=	0;
ePTO_OilRq_Tx.Data[3].0		:=	gq_ePTO_Activate;
ePTO_OilRq_Tx.Data[4]		:=	0;
ePTO_OilRq_Tx.Data[5]		:=	0;
ePTO_OilRq_Tx.Data[6]		:=	0;
ePTO_OilRq_Tx.Data[7]		:=	0;
ePTO_OilRq_Tx.Len			:=	8;
(**)


ePTO_Speed_47A_Tx.ID		:=	16#47A;
ePTO_Speed_47A_Tx.Data[0]	:=	UINT_TO_USINT(gu16_TrqHi);
ePTO_Speed_47A_Tx.Data[1]	:=	UINT_TO_USINT(SHR(gu16_TrqHi, 8));
ePTO_Speed_47A_Tx.Data[2]	:=	UINT_TO_USINT(gu16_Skai_SpeedTarget);
ePTO_Speed_47A_Tx.Data[3]	:=	UINT_TO_USINT(SHR(gu16_Skai_SpeedTarget, 8));
ePTO_Speed_47A_Tx.Data[4]	:=	(BOOL_TO_USINT(gq_ePTO_Activate) * 2);
ePTO_Speed_47A_Tx.Data[5]	:=	gu8_Asym_Limits + gu8_DIGITAL1;
ePTO_Speed_47A_Tx.Data[6]	:=	0;
ePTO_Speed_47A_Tx.Data[7]	:=	0;
ePTO_Speed_47A_Tx.Len		:=	8;
	 
ePTO_Torque_57A_Tx.ID		:=	16#57A;
ePTO_Torque_57A_Tx.Data[0]	:=	UINT_TO_USINT(gu16_TrqHi);
ePTO_Torque_57A_Tx.Data[1]	:=	UINT_TO_USINT(SHR(gu16_TrqHi, 8));
ePTO_Torque_57A_Tx.Data[2]	:=	UINT_TO_USINT(gu16_TrqLo);
ePTO_Torque_57A_Tx.Data[3]	:=	UINT_TO_USINT(SHR(gu16_TrqLo, 8));
ePTO_Torque_57A_Tx.Data[4]	:=	0;
ePTO_Torque_57A_Tx.Data[5]	:=	0;
ePTO_Torque_57A_Tx.Data[6]	:=	0;
ePTO_Torque_57A_Tx.Data[7]	:=	0;
ePTO_Torque_57A_Tx.Len		:=	8;

(*CANOpen*)
ePTO_NMT_Tx.ID				:=	16#00;
ePTO_NMT_Tx.Data[0]			:=	gu8_CANOpen_Command;
ePTO_NMT_Tx.Data[1]			:=	gu8_CANOpen_NodeAddress;
ePTO_NMT_Tx.Len				:=	8;
{endregion}

	 
(**************************************************************************************************************************************************)
{region "Send Messages"}
(*Transmit*)
hton_MercePTO_TxTimer(IN := NOT(hton_MercePTO_TxTimer.Q), PT := T#100MS);
IF (hton_MercePTO_TxTimer.Q = TRUE) THEN
	IF (gu8_ChassisType = CHASSIS_BOB OR gu8_ChassisType = CHASSIS_ESTARGLIDER) THEN
		G_CAN4_Channel.SendMessage(i_pMSG:=ADR(MercCurrentGear1_Tx)); 
		G_CAN4_Channel.SendMessage(i_pMSG:=ADR(MercLHFWheelSpd_Tx)); 
		G_CAN4_Channel.SendMessage(i_pMSG:=ADR(MercCurrentGear2_Tx)); 
		G_CAN4_Channel.SendMessage(i_pMSG:=ADR(MercControlRPM_Tx));
	ELSIF (gu8_ChassisType = CHASSIS_DENNIS) THEN
		;
	END_IF
 
	G_CAN4_Channel.SendMessage(i_pMSG:=ADR(ePTO_Speed_47A_Tx));
	G_CAN4_Channel.SendMessage(i_pMSG:=ADR(ePTO_Torque_57A_Tx)); 
	G_CAN4_Channel.SendMessage(i_pMSG:=ADR(ePTO_OilRq_Tx)); 
		 
	G_CAN4_Channel.SendMessage(i_pMSG:=ADR(ePTO_NMT_Tx)); 
END_IF

{end_region}

END_PROGRAM

// Application/UserCode/CAN3/CAN3_Tx
PROGRAM CAN3_Tx
VAR
	ht_Bob_Allison_ETC7_Tx		:	EPEC_CANVXD.Msg;
	ht_Allison_Override_Tx: EPEC_CANVXD.Msg;
	ht_Bob_Allison_ProbA_Tx		:	EPEC_CANVXD.Msg;
	hton_MessageSend_Timer		:	TON;
END_VAR



(*Allison Selector Return*)
ht_Bob_Allison_ETC7_Tx.ID		:=	16#18FE4AD3 OR EPEC_CANVXD.MASK_29BIT;
ht_Bob_Allison_ETC7_Tx.Data[0]	:=	16#03;
ht_Bob_Allison_ETC7_Tx.Data[1]	:=	gu8_ETC7_TransmissionEngaged_Tx;
ht_Bob_Allison_ETC7_Tx.Data[2]	:=	16#4F;
ht_Bob_Allison_ETC7_Tx.Data[3]	:=	16#E0;
ht_Bob_Allison_ETC7_Tx.Data[4]	:=	16#FF;
ht_Bob_Allison_ETC7_Tx.Data[5]	:=	16#F3;
ht_Bob_Allison_ETC7_Tx.Data[6]	:=	16#FF;
ht_Bob_Allison_ETC7_Tx.Data[7]	:=	16#FF;
ht_Bob_Allison_ETC7_Tx.Len		:=	8;

ht_Bob_Allison_ProbA_Tx.ID		:=	16#18EF0503 OR EPEC_CANVXD.MASK_29BIT;
ht_Bob_Allison_ProbA_Tx.Data[0]	:=	16#0A;
ht_Bob_Allison_ProbA_Tx.Data[1]	:=	16#FC;
ht_Bob_Allison_ProbA_Tx.Data[2]	:=	16#00;
ht_Bob_Allison_ProbA_Tx.Data[3]	:=	16#01;
ht_Bob_Allison_ProbA_Tx.Data[4]	:=	16#23;
ht_Bob_Allison_ProbA_Tx.Data[5]	:=	16#01;
ht_Bob_Allison_ProbA_Tx.Data[6]	:=	gu8_ProbA_GearSelected_Tx;
ht_Bob_Allison_ProbA_Tx.Data[7]	:=	gu8_ProbA_GearSelected_Tx;
ht_Bob_Allison_ProbA_Tx.Len		:=	8;

ht_Allison_Override_Tx.ID		:= 16#18FF0400 OR EPEC_CANVXD.MASK_29BIT;
(*ht_Allison_Override_Tx.Data[0]	:=
ht_Allison_Override_Tx.Data[1]	:=
ht_Allison_Override_Tx.Data[2]	:=
ht_Allison_Override_Tx.Data[3]	:=*)
ht_Allison_Override_Tx.Data[4].0	:=	gq_Gear_Neutral;
ht_Allison_Override_Tx.Data[4].1	:=	gq_Gear_Drive;
ht_Allison_Override_Tx.Data[4].2	:=	gq_Gear_Reverse;
(*ht_Allison_Override_Tx.Data[5]	:=
ht_Allison_Override_Tx.Data[6]	:=
ht_Allison_Override_Tx.Data[7]	:=*)
ht_Allison_Override_Tx.Len		:=	8;

(*Transmit these messages*)
hton_MessageSend_Timer(IN := NOT(hton_MessageSend_Timer.Q), PT := T#100MS);
IF (hton_MessageSend_Timer.Q = TRUE) THEN
	G_CAN3_Channel.SendMessage(i_pMSG:=ADR(ht_Bob_Allison_ETC7_Tx));
	G_CAN3_Channel.SendMessage(i_pMSG:=ADR(ht_Bob_Allison_ProbA_Tx));
END_IF

IF (hton_MessageSend_Timer.Q = TRUE AND gq_Allison_Pad_Override = TRUE) THEN
	G_CAN3_Channel.SendMessage(i_pMSG:=ADR(ht_Allison_Override_Tx));
END_IF

END_PROGRAM

// Application/UserCode/CAN1/KB_Tx
PROGRAM KB_Tx
VAR
	ht_ETC1_Tx		:	EPEC_CANVXD.Msg;
	ht_ETC2_Tx		:	EPEC_CANVXD.Msg;
	ht_ETC8_Tx		:	EPEC_CANVXD.Msg;
	ht_ERC1_RD_Tx	:	EPEC_CANVXD.Msg;
	ht_ERC1_RE_Tx	:	EPEC_CANVXD.Msg;
	ht_RC_RD_Tx		:	EPEC_CANVXD.Msg;
	ht_RC_RE_Tx		:	EPEC_CANVXD.Msg;
	ht_TD_Tx		:	EPEC_CANVXD.Msg;
	ht_Prop37_Tx	:	EPEC_CANVXD.Msg;
	ht_Prop40_Tx	:	EPEC_CANVXD.Msg;
	ht_Prop87_Tx	:	EPEC_CANVXD.Msg;
	
	hton_MessageSend_Timer	:	TON;
	hton_TD_Timer			:	TON;
END_VAR

ht_ETC1_Tx.ID		:=	16#0CF00203 OR EPEC_CANVXD.MASK_29BIT;
ht_ETC1_Tx.Data[0]	:=	16#3D;
ht_ETC1_Tx.Data[1]	:=	16#00;
ht_ETC1_Tx.Data[2]	:=	16#00;
ht_ETC1_Tx.Data[3]	:=	16#00;
ht_ETC1_Tx.Data[4]	:=	16#00;
ht_ETC1_Tx.Data[5]	:=	16#00;
ht_ETC1_Tx.Data[6]	:=	16#00;
ht_ETC1_Tx.Data[7]	:=	16#00;
ht_ETC1_Tx.Len		:=	8;
	 
ht_ETC2_Tx.ID		:=	16#18F00503 OR EPEC_CANVXD.MASK_29BIT;
ht_ETC2_Tx.Data[0]	:=	gu8_CurrentGear2; (*Current Gear2*)
ht_ETC2_Tx.Data[1]	:=	UINT_TO_USINT(gu16_CurrentGear); (*Current Gear LSB*)
ht_ETC2_Tx.Data[2]	:=	UINT_TO_USINT(SHR(gu16_CurrentGear, 8)); (*Current Gear MSB*)
ht_ETC2_Tx.Data[3]	:=	gu8_CurrentGear2; (*Current Gear2*)
ht_ETC2_Tx.Data[4]	:=	16#FF;
ht_ETC2_Tx.Data[5]	:=	16#FF;
ht_ETC2_Tx.Data[6]	:=	UINT_TO_USINT(gu16_CurrentGear1); (*Current Gear1 LSB*)
ht_ETC2_Tx.Data[7]	:=	UINT_TO_USINT(SHR(gu16_CurrentGear1, 8)); (*Current Gear1 MSB*)
ht_ETC2_Tx.Len		:=	8;

ht_ETC8_Tx.ID		:=	16#0CF00C03 OR EPEC_CANVXD.MASK_29BIT;
ht_ETC8_Tx.Data[0]	:=	16#FF;
ht_ETC8_Tx.Data[1]	:=	16#FF;
ht_ETC8_Tx.Data[2]	:=	16#FF;
ht_ETC8_Tx.Data[3]	:=	16#FF;
ht_ETC8_Tx.Data[4]	:=	16#FF;
ht_ETC8_Tx.Data[5]	:=	16#FF;
ht_ETC8_Tx.Data[6]	:=	16#FF;
ht_ETC8_Tx.Data[7]	:=	16#FF;
ht_ETC8_Tx.Len		:=	8;

ht_ERC1_RD_Tx.ID		:=	16#18F00010 OR EPEC_CANVXD.MASK_29BIT;
ht_ERC1_RD_Tx.Data[0]	:=	16#00;
ht_ERC1_RD_Tx.Data[1]	:=	16#00;
ht_ERC1_RD_Tx.Data[2]	:=	16#00;
ht_ERC1_RD_Tx.Data[3]	:=	16#00;
ht_ERC1_RD_Tx.Data[4]	:=	16#00;
ht_ERC1_RD_Tx.Data[5]	:=	16#00;
ht_ERC1_RD_Tx.Data[6]	:=	16#00;
ht_ERC1_RD_Tx.Data[7]	:=	16#A5;
ht_ERC1_RD_Tx.Len		:=	8;

ht_ERC1_RE_Tx.ID		:=	16#18F0000F OR EPEC_CANVXD.MASK_29BIT;
ht_ERC1_RE_Tx.Data[0]	:=	16#00;
ht_ERC1_RE_Tx.Data[1]	:=	16#A5;
ht_ERC1_RE_Tx.Data[2]	:=	16#00;
ht_ERC1_RE_Tx.Data[3]	:=	16#00;
ht_ERC1_RE_Tx.Data[4]	:=	16#00;
ht_ERC1_RE_Tx.Data[5]	:=	16#00;
ht_ERC1_RE_Tx.Data[6]	:=	16#00;
ht_ERC1_RE_Tx.Data[7]	:=	16#A5;
ht_ERC1_RE_Tx.Len		:=	8;

ht_RC_RD_Tx.ID		:=	16#18FEE110 OR EPEC_CANVXD.MASK_29BIT;
ht_RC_RD_Tx.Data[0]	:=	16#00;
ht_RC_RD_Tx.Data[1]	:=	16#10;
ht_RC_RD_Tx.Data[2]	:=	16#00;
ht_RC_RD_Tx.Data[3]	:=	16#00;
ht_RC_RD_Tx.Data[4]	:=	16#00;
ht_RC_RD_Tx.Data[5]	:=	16#00;
ht_RC_RD_Tx.Data[6]	:=	16#00;
ht_RC_RD_Tx.Data[7]	:=	16#00;
ht_RC_RD_Tx.Len		:=	8;

ht_RC_RE_Tx.ID		:=	16#18FEE10F OR EPEC_CANVXD.MASK_29BIT;
ht_RC_RE_Tx.Data[0]	:=	16#00;
ht_RC_RE_Tx.Data[1]	:=	16#00;
ht_RC_RE_Tx.Data[2]	:=	16#FF;
ht_RC_RE_Tx.Data[3]	:=	16#FF;
ht_RC_RE_Tx.Data[4]	:=	16#FF;
ht_RC_RE_Tx.Data[5]	:=	16#FF;
ht_RC_RE_Tx.Data[6]	:=	16#FF;
ht_RC_RE_Tx.Data[7]	:=	16#FF;
ht_RC_RE_Tx.Len		:=	8;

ht_TD_Tx.ID			:=	16#18FEE617 OR EPEC_CANVXD.MASK_29BIT;
ht_TD_Tx.Data[0]	:=	16#FF;
ht_TD_Tx.Data[1]	:=	16#FF;
ht_TD_Tx.Data[2]	:=	16#FF;
ht_TD_Tx.Data[3]	:=	16#FF;
ht_TD_Tx.Data[4]	:=	16#FF;
ht_TD_Tx.Data[5]	:=	16#FF;
ht_TD_Tx.Data[6]	:=	16#00;
ht_TD_Tx.Data[7]	:=	16#00;
ht_TD_Tx.Len		:=	8;

ht_Prop37_Tx.ID			:=	16#0CFF2537 OR EPEC_CANVXD.MASK_29BIT;
ht_Prop37_Tx.Data[0]	:=	16#FF;
ht_Prop37_Tx.Data[1]	:=	16#FF;
ht_Prop37_Tx.Data[2]	:=	16#00;
ht_Prop37_Tx.Data[3]	:=	16#00;
ht_Prop37_Tx.Data[4]	:=	16#00;
ht_Prop37_Tx.Data[5]	:=	16#00;
ht_Prop37_Tx.Data[6]	:=	16#00;
ht_Prop37_Tx.Data[7]	:=	16#FC;
ht_Prop37_Tx.Len		:=	8;

ht_Prop40_Tx.ID			:=	16#0CFF2817 OR EPEC_CANVXD.MASK_29BIT;
ht_Prop40_Tx.Data[0]	:=	16#FC;
ht_Prop40_Tx.Data[1]	:=	16#F3;
ht_Prop40_Tx.Data[2]	:=	16#FF;
ht_Prop40_Tx.Data[3]	:=	16#00;
ht_Prop40_Tx.Data[4]	:=	16#00;
ht_Prop40_Tx.Data[5]	:=	16#00;
ht_Prop40_Tx.Data[6]	:=	16#00;
ht_Prop40_Tx.Data[7]	:=	16#00;
ht_Prop40_Tx.Len		:=	8;

ht_Prop87_Tx.ID			:=	16#0CFF5730 OR EPEC_CANVXD.MASK_29BIT;
ht_Prop87_Tx.Data[0]	:=	16#FF;
ht_Prop87_Tx.Data[1]	:=	16#FD;
ht_Prop87_Tx.Data[2]	:=	16#00;
ht_Prop87_Tx.Data[3]	:=	16#00;
ht_Prop87_Tx.Data[4]	:=	16#00;
ht_Prop87_Tx.Data[5]	:=	16#00;
ht_Prop87_Tx.Data[6]	:=	16#00;
ht_Prop87_Tx.Data[7]	:=	16#00;
ht_Prop87_Tx.Len		:=	8;




hton_MessageSend_Timer(IN := NOT(hton_MessageSend_Timer.Q), PT := T#80MS);
IF (hton_MessageSend_Timer.Q = TRUE) THEN
	G_CAN1_Channel.SendMessage(i_pMSG:=ADR(ht_ETC1_Tx));
	G_CAN1_Channel.SendMessage(i_pMSG:=ADR(ht_ETC2_Tx));
	G_CAN1_Channel.SendMessage(i_pMSG:=ADR(ht_ETC8_Tx));
	G_CAN1_Channel.SendMessage(i_pMSG:=ADR(ht_ERC1_RD_Tx));
	G_CAN1_Channel.SendMessage(i_pMSG:=ADR(ht_ERC1_RE_Tx));
	G_CAN1_Channel.SendMessage(i_pMSG:=ADR(ht_RC_RD_Tx));
	G_CAN1_Channel.SendMessage(i_pMSG:=ADR(ht_RC_RE_Tx));
	G_CAN1_Channel.SendMessage(i_pMSG:=ADR(ht_Prop37_Tx));
	G_CAN1_Channel.SendMessage(i_pMSG:=ADR(ht_Prop40_Tx));
	G_CAN1_Channel.SendMessage(i_pMSG:=ADR(ht_Prop87_Tx));
END_IF

hton_TD_Timer(IN := NOT(hton_TD_Timer.Q), PT := T#10000MS);
IF (hton_TD_Timer.Q = TRUE) THEN
	G_CAN1_Channel.SendMessage(i_pMSG:=ADR(ht_TD_Tx));
END_IF

END_PROGRAM

// Application/UserCode/CAN1/CAN1_TCMs_Tx
PROGRAM CAN1_TCMs_Tx
VAR
	(*TCM ECR*)
	ht_RCM_C01_Tx	:	EPEC_CANVXD.Msg;
	ht_RCM_C02_Tx	:	EPEC_CANVXD.Msg;
	ht_TCM_C01_Tx	:	EPEC_CANVXD.Msg;
	ht_TCM_C02_Tx	:	EPEC_CANVXD.Msg;
	ht_TCM_C03_Tx	:	EPEC_CANVXD.Msg;
	ht_TCM_C05_Tx	:	EPEC_CANVXD.Msg;
	ht_TCM_C06_Tx	:	EPEC_CANVXD.Msg;
	ht_TCM_C08_Tx	:	EPEC_CANVXD.Msg;
	ht_TCM_C10_Tx	:	EPEC_CANVXD.Msg;
	ht_TCM_C11_Tx	:	EPEC_CANVXD.Msg;
	ht_TCM_C22_Tx	:	EPEC_CANVXD.Msg;
	ht_TCM_DM1_Tx	:	EPEC_CANVXD.Msg;
	ht_TRF1_TCM_Tx	:	EPEC_CANVXD.Msg;
	
	ht_MCM_C01_Tx	:	EPEC_CANVXD.Msg;
	ht_MCM_C02_Tx	:	EPEC_CANVXD.Msg;
	ht_MCM_C03_Tx	:	EPEC_CANVXD.Msg;
	ht_MCM_C07_Tx	:	EPEC_CANVXD.Msg;
	ht_MCM_C10_Tx	:	EPEC_CANVXD.Msg;
	ht_MCM_C14_Tx	:	EPEC_CANVXD.Msg;
	ht_MCM_C15_Tx	:	EPEC_CANVXD.Msg;
	ht_MCM_C23_Tx	:	EPEC_CANVXD.Msg;
	
	ht_Compressor_Status	:	EPEC_CANVXD.Msg;
	
	hu8_C01_Checksum	:	USINT;
	hu8_C02_Checksum	:	USINT;
	hu8_C03_Checksum	:	USINT;
	hu8_C05_Checksum	:	USINT;
	hu8_C08_Checksum	:	USINT;
	hu8_C10_Checksum	:	USINT;
	hu8_C11_Checksum	:	USINT;
	hu8_M23_Checksum	:	USINT;
	
	hu8_4BitMessageCounter10ms		:	USINT;
	hu8_4BitMessageCounter20ms		:	USINT;
	hu8_4BitMessageCounter50ms		:	USINT;
	hu8_4BitMessageCounter100ms		:	USINT;
	
	hq_CycleAlternator	:	BOOL;
	hton_MessageSend50ms_Timer	:	TON;
	hton_MessageSend_Timer		:	TON;
	Tx_Timer	:	TON;
	ClutchEnaged: BOOL;
END_VAR
VAR CONSTANT
	MAX_REGEN_TORQUE	:	UINT	:=	4090;
END_VAR
VAR
	ClutchStatB: BOOL := TRUE;
	ClutchStatA: BOOL := TRUE;
	ClutchEngaged: BOOL;
	ClutchIntermediate: BOOL;
	ClutchDisengaged: BOOL;
	TONIntermediate: TON;
END_VAR

ht_RCM_C01_Tx.ID		:=	16#CFF000F OR EPEC_CANVXD.MASK_29BIT;
ht_RCM_C01_Tx.Data[0]	:=	16#FF;
ht_RCM_C01_Tx.Data[1].0	:=	gq_RegenActive;
ht_RCM_C01_Tx.Data[1].1	:=	0;
ht_RCM_C01_Tx.Data[1].2	:=	gq_RegenActive;
ht_RCM_C01_Tx.Data[1].3	:=	0;
ht_RCM_C01_Tx.Data[1].4	:=	1;
ht_RCM_C01_Tx.Data[1].5	:=	1;
ht_RCM_C01_Tx.Data[1].6	:=	1;
ht_RCM_C01_Tx.Data[1].7	:=	1;
ht_RCM_C01_Tx.Data[2]	:=	16#FF;
ht_RCM_C01_Tx.Data[3]	:=	REAL_TO_USINT(ABS(MIN(0, gr_MCU_TorqueCommand_PreCF * BOOL_TO_USINT(gq_RegenActive) / 20))); //Should be 0 when not regenning and then a positive value when it is doing so
ht_RCM_C01_Tx.Data[4]	:=	REAL_TO_USINT(MAX_REGEN_TORQUE / 20); //Maximum regen torque is 4090Nm (MCU CAN Protocol v4.1)
ht_RCM_C01_Tx.Data[5]	:=	16#FF;
ht_RCM_C01_Tx.Data[6]	:=	16#FF;
ht_RCM_C01_Tx.Data[7]	:=	16#FF;
ht_RCM_C01_Tx.Len		:=	8;
	 
ht_RCM_C02_Tx.ID		:=	16#14FF000F OR EPEC_CANVXD.MASK_29BIT;
ht_RCM_C02_Tx.Data[0]	:=	16#FF;
ht_RCM_C02_Tx.Data[1]	:=	16#FF;
ht_RCM_C02_Tx.Data[2]	:=	16#FF;
ht_RCM_C02_Tx.Data[3]	:=	16#FF;
ht_RCM_C02_Tx.Data[4]	:=	16#FF;
ht_RCM_C02_Tx.Data[5]	:=	16#FF;
ht_RCM_C02_Tx.Data[6]	:=	16#FF;
ht_RCM_C02_Tx.Data[7]	:=	16#FF;
ht_RCM_C02_Tx.Len		:=	8;
	 
ht_TCM_C01_Tx.ID		:=	16#08FF0003 OR EPEC_CANVXD.MASK_29BIT;
ht_TCM_C01_Tx.Data[0]	:=	16#FF;
ht_TCM_C01_Tx.Data[1]	:=	16#FF;
ht_TCM_C01_Tx.Data[2]	:=	16#FF;
ht_TCM_C01_Tx.Data[3]	:=	16#FF;
ht_TCM_C01_Tx.Data[4]	:=	16#FF;
ht_TCM_C01_Tx.Data[5]	:=	16#FF;
ht_TCM_C01_Tx.Data[6].0	:=	1;
ht_TCM_C01_Tx.Data[6].1	:=	1;
ht_TCM_C01_Tx.Data[6].2	:=	1;
ht_TCM_C01_Tx.Data[6].3	:=	1;
ht_TCM_C01_Tx.Data[6].4	:=	hu8_4BitMessageCounter10ms.0;
ht_TCM_C01_Tx.Data[6].5	:=	hu8_4BitMessageCounter10ms.1;
ht_TCM_C01_Tx.Data[6].6	:=	hu8_4BitMessageCounter10ms.2;
ht_TCM_C01_Tx.Data[6].7	:=	hu8_4BitMessageCounter10ms.3;
hu8_C01_Checksum		:=	16#FF - (ht_TCM_C01_Tx.Data[0] + ht_TCM_C01_Tx.Data[1] + ht_TCM_C01_Tx.Data[2] + ht_TCM_C01_Tx.Data[3] + ht_TCM_C01_Tx.Data[4] + ht_TCM_C01_Tx.Data[5] + ht_TCM_C01_Tx.Data[6]);;
ht_TCM_C01_Tx.Data[7]	:=	hu8_C01_Checksum;
ht_TCM_C01_Tx.Len		:=	8;

ht_TCM_C02_Tx.ID		:=	16#08FF0103 OR EPEC_CANVXD.MASK_29BIT;
ht_TCM_C02_Tx.Data[0]	:=	16#FF;
ht_TCM_C02_Tx.Data[1]	:=	16#FF;
ht_TCM_C02_Tx.Data[2]	:=	UINT_TO_USINT(gu16_TCM2_OutputShaftSpeed);
ht_TCM_C02_Tx.Data[3]	:=	UINT_TO_USINT(SHR(gu16_TCM2_OutputShaftSpeed, 8));
ht_TCM_C02_Tx.Data[4]	:=	16#FF;
ht_TCM_C02_Tx.Data[5].0	:=	gu8_TCM2_DrvDirec_Stat.0;
ht_TCM_C02_Tx.Data[5].1	:=	gu8_TCM2_DrvDirec_Stat.1;
ht_TCM_C02_Tx.Data[5].2	:=	1;
ht_TCM_C02_Tx.Data[5].3	:=	1;
ht_TCM_C02_Tx.Data[5].4	:=	gu8_TCM2_RotSens_Stat.0;
ht_TCM_C02_Tx.Data[5].5	:=	gu8_TCM2_RotSens_Stat.1;
ht_TCM_C02_Tx.Data[5].6	:=	1;
ht_TCM_C02_Tx.Data[5].7	:=	1;
ht_TCM_C02_Tx.Data[6].0	:=	ClutchStatA;
ht_TCM_C02_Tx.Data[6].1	:=	ClutchStatB;
ht_TCM_C02_Tx.Data[6].2	:=	1;
ht_TCM_C02_Tx.Data[6].3	:=	1;
ht_TCM_C02_Tx.Data[6].4	:=	hu8_4BitMessageCounter10ms.0;
ht_TCM_C02_Tx.Data[6].5	:=	hu8_4BitMessageCounter10ms.1;
ht_TCM_C02_Tx.Data[6].6	:=	hu8_4BitMessageCounter10ms.2;
ht_TCM_C02_Tx.Data[6].7	:=	hu8_4BitMessageCounter10ms.3;
hu8_C02_Checksum	:=	16#FF - (ht_TCM_C02_Tx.Data[0] + ht_TCM_C02_Tx.Data[1] + ht_TCM_C02_Tx.Data[2] + ht_TCM_C02_Tx.Data[3] + ht_TCM_C02_Tx.Data[4] + ht_TCM_C02_Tx.Data[5] + ht_TCM_C02_Tx.Data[6]);
ht_TCM_C02_Tx.Data[7]	:=	hu8_C02_Checksum;
ht_TCM_C02_Tx.Len		:=	8;

ht_TCM_C03_Tx.ID		:=	16#08FF0203 OR EPEC_CANVXD.MASK_29BIT;
ht_TCM_C03_Tx.Data[0]	:=	16#FF;
ht_TCM_C03_Tx.Data[1]	:=	16#FF;
ht_TCM_C03_Tx.Data[2]	:=	UINT_TO_USINT(gu16_TCM03_ShaftSpeed_Tx);
ht_TCM_C03_Tx.Data[3]	:=	UINT_TO_USINT(SHR(gu16_TCM03_ShaftSpeed_Tx, 8));
ht_TCM_C03_Tx.Data[4]	:=	16#FF;
ht_TCM_C03_Tx.Data[5]	:=	16#FF;
ht_TCM_C03_Tx.Data[6].0	:=	1;
ht_TCM_C03_Tx.Data[6].1	:=	1;
ht_TCM_C03_Tx.Data[6].2	:=	1;
ht_TCM_C03_Tx.Data[6].3	:=	1;
ht_TCM_C03_Tx.Data[6].4	:=	hu8_4BitMessageCounter10ms.0;
ht_TCM_C03_Tx.Data[6].5	:=	hu8_4BitMessageCounter10ms.1;
ht_TCM_C03_Tx.Data[6].6	:=	hu8_4BitMessageCounter10ms.2;
ht_TCM_C03_Tx.Data[6].7	:=	hu8_4BitMessageCounter10ms.3;
hu8_C03_Checksum	:=	16#FF - (ht_TCM_C03_Tx.Data[0] + ht_TCM_C03_Tx.Data[1] + ht_TCM_C03_Tx.Data[2] + ht_TCM_C03_Tx.Data[3] + ht_TCM_C03_Tx.Data[4] + ht_TCM_C03_Tx.Data[5] + ht_TCM_C03_Tx.Data[6]);
ht_TCM_C03_Tx.Data[7]	:=	hu8_C03_Checksum;
ht_TCM_C03_Tx.Len		:=	8;

ht_TCM_C05_Tx.ID		:=	16#14FF0403 OR EPEC_CANVXD.MASK_29BIT;
ht_TCM_C05_Tx.Data[0]	:=	16#FF;
ht_TCM_C05_Tx.Data[1]	:=	16#FF;
ht_TCM_C05_Tx.Data[2]	:=	16#FF;
ht_TCM_C05_Tx.Data[3]	:=	16#FF;
ht_TCM_C05_Tx.Data[4]	:=	16#FF;
ht_TCM_C05_Tx.Data[5]	:=	16#FF;
ht_TCM_C05_Tx.Data[6].0	:=	gq_Gear_Neutral;
ht_TCM_C05_Tx.Data[6].1	:=	0;
ht_TCM_C05_Tx.Data[6].2	:=	1;
ht_TCM_C05_Tx.Data[6].3	:=	1;
ht_TCM_C05_Tx.Data[6].4	:=	hu8_4BitMessageCounter100ms.0;
ht_TCM_C05_Tx.Data[6].5	:=	hu8_4BitMessageCounter100ms.1;
ht_TCM_C05_Tx.Data[6].6	:=	hu8_4BitMessageCounter100ms.2;
ht_TCM_C05_Tx.Data[6].7	:=	hu8_4BitMessageCounter100ms.3;
hu8_C05_Checksum	:=	16#FF - (ht_TCM_C05_Tx.Data[0] + ht_TCM_C05_Tx.Data[1] + ht_TCM_C05_Tx.Data[2] + ht_TCM_C05_Tx.Data[3] + ht_TCM_C05_Tx.Data[4] + ht_TCM_C05_Tx.Data[5] + ht_TCM_C05_Tx.Data[6]);
ht_TCM_C05_Tx.Data[7]	:=	hu8_C05_Checksum;
ht_TCM_C05_Tx.Len		:=	8;

ht_TCM_C06_Tx.ID		:=	16#18FF0503 OR EPEC_CANVXD.MASK_29BIT;
ht_TCM_C06_Tx.Data[0]	:=	16#FF;
ht_TCM_C06_Tx.Data[1]	:=	16#FF;
ht_TCM_C06_Tx.Data[2]	:=	16#FF;
ht_TCM_C06_Tx.Data[3]	:=	16#FF;
ht_TCM_C06_Tx.Data[4]	:=	16#FF;
ht_TCM_C06_Tx.Data[5]	:=	16#FF;
ht_TCM_C06_Tx.Data[6]	:=	16#FF;
ht_TCM_C06_Tx.Data[7]	:=	16#FF;
ht_TCM_C06_Tx.Len		:=	8;

ht_TCM_C08_Tx.ID		:=	16#0CFF0703 OR EPEC_CANVXD.MASK_29BIT;
ht_TCM_C08_Tx.Data[0]	:=	16#FF;
ht_TCM_C08_Tx.Data[1]	:=	16#FF;
ht_TCM_C08_Tx.Data[2]	:=	16#FF;
ht_TCM_C08_Tx.Data[3]	:=	16#FF;
ht_TCM_C08_Tx.Data[4]	:=	gu8_TCM8_Gear;
ht_TCM_C08_Tx.Data[5]	:=	16#FF;
ht_TCM_C08_Tx.Data[6].0	:=	NOT(gq_Gear_Neutral);
ht_TCM_C08_Tx.Data[6].1	:=	0;
ht_TCM_C08_Tx.Data[6].2	:=	gu8_TCM8_DrvDirByGr_Stat.0;
ht_TCM_C08_Tx.Data[6].3	:=	gu8_TCM8_DrvDirByGr_Stat.1;
ht_TCM_C08_Tx.Data[6].4	:=	hu8_4BitMessageCounter20ms.0;
ht_TCM_C08_Tx.Data[6].5	:=	hu8_4BitMessageCounter20ms.1;
ht_TCM_C08_Tx.Data[6].6	:=	hu8_4BitMessageCounter20ms.2;
ht_TCM_C08_Tx.Data[6].7	:=	hu8_4BitMessageCounter20ms.3;
hu8_C08_Checksum	:=	16#FF - (ht_TCM_C08_Tx.Data[0] + ht_TCM_C08_Tx.Data[1] + ht_TCM_C08_Tx.Data[2] + ht_TCM_C08_Tx.Data[3] + ht_TCM_C08_Tx.Data[4] + ht_TCM_C08_Tx.Data[5] + ht_TCM_C08_Tx.Data[6]);
ht_TCM_C08_Tx.Data[7]	:=	hu8_C08_Checksum;
ht_TCM_C08_Tx.Len		:=	8;

ht_TCM_C10_Tx.ID		:=	16#10FF0903 OR EPEC_CANVXD.MASK_29BIT;
ht_TCM_C10_Tx.Data[0]	:=	16#FF;
ht_TCM_C10_Tx.Data[1]	:=	16#FF;
ht_TCM_C10_Tx.Data[2]	:=	16#FF;
ht_TCM_C10_Tx.Data[3]	:=	16#FF;
ht_TCM_C10_Tx.Data[4]	:=	16#FF;
ht_TCM_C10_Tx.Data[5]	:=	16#FF;
ht_TCM_C10_Tx.Data[6].0	:=	1;
ht_TCM_C10_Tx.Data[6].1	:=	1;
ht_TCM_C10_Tx.Data[6].2	:=	1;
ht_TCM_C10_Tx.Data[6].3	:=	1;
ht_TCM_C10_Tx.Data[6].4	:=	hu8_4BitMessageCounter50ms.0;
ht_TCM_C10_Tx.Data[6].5	:=	hu8_4BitMessageCounter50ms.1;
ht_TCM_C10_Tx.Data[6].6	:=	hu8_4BitMessageCounter50ms.2;
ht_TCM_C10_Tx.Data[6].7	:=	hu8_4BitMessageCounter50ms.3;
hu8_C10_Checksum	:=	16#FF - (ht_TCM_C10_Tx.Data[0] + ht_TCM_C10_Tx.Data[1] + ht_TCM_C10_Tx.Data[2] + ht_TCM_C10_Tx.Data[3] + ht_TCM_C10_Tx.Data[4] + ht_TCM_C10_Tx.Data[5] + ht_TCM_C10_Tx.Data[6]);
ht_TCM_C10_Tx.Data[7]	:=	0;
ht_TCM_C10_Tx.Len		:=	8;

ht_TCM_C11_Tx.ID		:=	16#08FF0303 OR EPEC_CANVXD.MASK_29BIT;
ht_TCM_C11_Tx.Data[0]	:=	gu8_TCM8_Gear;
ht_TCM_C11_Tx.Data[1]	:=	16#FF;
ht_TCM_C11_Tx.Data[2]	:=	16#FF;
ht_TCM_C11_Tx.Data[3]	:=	16#FF;
ht_TCM_C11_Tx.Data[4]	:=	16#FF;
ht_TCM_C11_Tx.Data[5]	:=	16#FF;
ht_TCM_C11_Tx.Data[6]	:=	UINT_TO_USINT(gu16_TCM11_ActualGearRatio);
ht_TCM_C11_Tx.Data[7]	:=	UINT_TO_USINT(SHR(gu16_TCM11_ActualGearRatio, 8));
ht_TCM_C11_Tx.Len		:=	8;

ht_TCM_C22_Tx.ID		:=	16#18FF0703 OR EPEC_CANVXD.MASK_29BIT;
ht_TCM_C22_Tx.Data[0]	:=	16#FF;
ht_TCM_C22_Tx.Data[1]	:=	16#FF;
ht_TCM_C22_Tx.Data[2]	:=	16#FF;
ht_TCM_C22_Tx.Data[3]	:=	16#FF;
ht_TCM_C22_Tx.Data[4]	:=	16#FF;
ht_TCM_C22_Tx.Data[5]	:=	16#FF;
ht_TCM_C22_Tx.Data[6]	:=	16#FF;
ht_TCM_C22_Tx.Data[7]	:=	16#FF;
ht_TCM_C22_Tx.Len		:=	8;

(*Message not sent*)
ht_TCM_DM1_Tx.ID		:=	16#10FECA03 OR EPEC_CANVXD.MASK_29BIT;
ht_TCM_DM1_Tx.Data[0]	:=	0;
ht_TCM_DM1_Tx.Data[1]	:=	0;
ht_TCM_DM1_Tx.Data[2]	:=	0;
ht_TCM_DM1_Tx.Data[3]	:=	0;
ht_TCM_DM1_Tx.Data[4]	:=	0;
ht_TCM_DM1_Tx.Data[5]	:=	0;
ht_TCM_DM1_Tx.Data[6]	:=	0;
ht_TCM_DM1_Tx.Data[7]	:=	0;
ht_TCM_DM1_Tx.Len		:=	8;

ht_TRF1_TCM_Tx.ID		:=	16#18FEF803 OR EPEC_CANVXD.MASK_29BIT;
ht_TRF1_TCM_Tx.Data[0]	:=	16#FF;
ht_TRF1_TCM_Tx.Data[1]	:=	16#FF;
ht_TRF1_TCM_Tx.Data[2]	:=	16#FF;
ht_TRF1_TCM_Tx.Data[3]	:=	16#FF;
ht_TRF1_TCM_Tx.Data[4]	:=	16#FF;
ht_TRF1_TCM_Tx.Data[5]	:=	16#FF;
ht_TRF1_TCM_Tx.Data[6]	:=	16#FF;
ht_TRF1_TCM_Tx.Data[7]	:=	16#FF;
ht_TRF1_TCM_Tx.Len		:=	8;

(*********************************************************************)
ht_MCM_C01_Tx.ID		:=	16#08FF0001 OR EPEC_CANVXD.MASK_29BIT;
ht_MCM_C01_Tx.Data[0]	:=	16#FF;
ht_MCM_C01_Tx.Data[1]	:=	16#FF;
ht_MCM_C01_Tx.Data[2]	:=	16#FF;
ht_MCM_C01_Tx.Data[3]	:=	16#FF;
ht_MCM_C01_Tx.Data[4]	:=	16#FF;
ht_MCM_C01_Tx.Data[5]	:=	16#FF;
ht_MCM_C01_Tx.Data[6]	:=	16#FF;
ht_MCM_C01_Tx.Data[7]	:=	16#FF;
ht_MCM_C01_Tx.Len		:=	8;

ht_MCM_C02_Tx.ID		:=	16#08FF0101 OR EPEC_CANVXD.MASK_29BIT; (*commented out due to already being sent*)
ht_MCM_C02_Tx.Data[0]	:=	BOOL_TO_USINT(DOS_q_BatteryDischargeMain_DO);
ht_MCM_C02_Tx.Data[1]	:=	16#FF;
ht_MCM_C02_Tx.Data[2]	:=	UINT_TO_USINT(gu16_MCM02_EngineTorque_Tx);
ht_MCM_C02_Tx.Data[3]	:=	UINT_TO_USINT(SHR(gu16_MCM02_EngineTorque_Tx, 8));
ht_MCM_C02_Tx.Data[4]	:=	UINT_TO_USINT(gu16_RPM_Display);
ht_MCM_C02_Tx.Data[5]	:=	UINT_TO_USINT(SHR(gu16_RPM_Display, 8));
ht_MCM_C02_Tx.Data[6]	:=	16#FF;
ht_MCM_C02_Tx.Data[7]	:=	16#FF;
ht_MCM_C02_Tx.Len		:=	8;

ht_MCM_C03_Tx.ID		:=	16#14FF0001 OR EPEC_CANVXD.MASK_29BIT;
ht_MCM_C03_Tx.Data[0]	:=	16#FF;
ht_MCM_C03_Tx.Data[1]	:=	16#FF;
ht_MCM_C03_Tx.Data[2]	:=	16#FF;
ht_MCM_C03_Tx.Data[3]	:=	16#FF;
ht_MCM_C03_Tx.Data[4]	:=	16#FF;
ht_MCM_C03_Tx.Data[5]	:=	16#FF;
ht_MCM_C03_Tx.Data[6]	:=	16#FF;
ht_MCM_C03_Tx.Data[7]	:=	16#FF;
ht_MCM_C03_Tx.Len		:=	8;

ht_MCM_C07_Tx.ID		:=	16#14FF0401 OR EPEC_CANVXD.MASK_29BIT;
ht_MCM_C07_Tx.Data[0]	:=	16#FF;
ht_MCM_C07_Tx.Data[1]	:=	16#FF;
ht_MCM_C07_Tx.Data[2]	:=	16#FF;
ht_MCM_C07_Tx.Data[3]	:=	16#FF;
ht_MCM_C07_Tx.Data[4]	:=	16#FF;
ht_MCM_C07_Tx.Data[5]	:=	16#FF;
ht_MCM_C07_Tx.Data[6]	:=	16#FF;
ht_MCM_C07_Tx.Data[7]	:=	16#FF;
ht_MCM_C07_Tx.Len		:=	8;

ht_MCM_C10_Tx.ID		:=	16#18FF0201 OR EPEC_CANVXD.MASK_29BIT;
ht_MCM_C10_Tx.Data[0]	:=	16#FF;
ht_MCM_C10_Tx.Data[1]	:=	16#FF;
ht_MCM_C10_Tx.Data[2]	:=	16#FF;
ht_MCM_C10_Tx.Data[3]	:=	16#FF;
ht_MCM_C10_Tx.Data[4]	:=	16#FF;
ht_MCM_C10_Tx.Data[5]	:=	16#FF;
ht_MCM_C10_Tx.Data[6]	:=	16#FF;
ht_MCM_C10_Tx.Data[7]	:=	16#FF;
ht_MCM_C10_Tx.Len		:=	8;

ht_MCM_C14_Tx.ID		:=	16#18FF0401 OR EPEC_CANVXD.MASK_29BIT;
ht_MCM_C14_Tx.Data[0]	:=	16#FF;
ht_MCM_C14_Tx.Data[1]	:=	16#FF;
ht_MCM_C14_Tx.Data[2]	:=	16#FF;
ht_MCM_C14_Tx.Data[3]	:=	16#FF;
ht_MCM_C14_Tx.Data[4]	:=	16#FF;
ht_MCM_C14_Tx.Data[5]	:=	16#FF;
ht_MCM_C14_Tx.Data[6]	:=	16#FF;
ht_MCM_C14_Tx.Data[7]	:=	16#FF;
ht_MCM_C14_Tx.Len		:=	8;

ht_MCM_C15_Tx.ID		:=	16#0CFF0001 OR EPEC_CANVXD.MASK_29BIT;
ht_MCM_C15_Tx.Data[0]	:=	16#FF;
ht_MCM_C15_Tx.Data[1]	:=	16#FF;
ht_MCM_C15_Tx.Data[2]	:=	16#FF;
ht_MCM_C15_Tx.Data[3]	:=	16#FF;
ht_MCM_C15_Tx.Data[4]	:=	16#FF;
ht_MCM_C15_Tx.Data[5]	:=	16#FF;
ht_MCM_C15_Tx.Data[6]	:=	16#FF;
ht_MCM_C15_Tx.Data[7]	:=	16#FF;
ht_MCM_C15_Tx.Len		:=	8;

ht_MCM_C23_Tx.ID		:=	16#08FF0201 OR EPEC_CANVXD.MASK_29BIT;
ht_MCM_C23_Tx.Data[0]	:=	16#FF;
ht_MCM_C23_Tx.Data[1]	:=	16#FF;
ht_MCM_C23_Tx.Data[2]	:=	16#FF;
ht_MCM_C23_Tx.Data[3]	:=	16#FF;
ht_MCM_C23_Tx.Data[4]	:=	16#FF;
ht_MCM_C23_Tx.Data[5]	:=	16#FF;
ht_MCM_C23_Tx.Data[6].0	:=	1;
ht_MCM_C23_Tx.Data[6].1	:=	1;
ht_MCM_C23_Tx.Data[6].2	:=	1;
ht_MCM_C23_Tx.Data[6].3	:=	1;
ht_MCM_C23_Tx.Data[6].4	:=	hu8_4BitMessageCounter10ms.0;
ht_MCM_C23_Tx.Data[6].5	:=	hu8_4BitMessageCounter10ms.1;
ht_MCM_C23_Tx.Data[6].6	:=	hu8_4BitMessageCounter10ms.2;
ht_MCM_C23_Tx.Data[6].7	:=	hu8_4BitMessageCounter10ms.3;
hu8_M23_Checksum	:=	16#FF - (ht_MCM_C23_Tx.Data[0] + ht_MCM_C23_Tx.Data[1] + ht_MCM_C23_Tx.Data[2] + ht_MCM_C23_Tx.Data[3] + ht_MCM_C23_Tx.Data[4] + ht_MCM_C23_Tx.Data[5] + ht_MCM_C23_Tx.Data[6]);
ht_MCM_C23_Tx.Data[7]	:=	hu8_M23_Checksum;
ht_MCM_C23_Tx.Len		:=	8;

(*Return status of the AIR1 message to inform the chassis if the compressor is on or off DAIMLER chassis
ht_Compressor_Status.ID	:=	16#14FEAE8C OR EPEC_CANVXD.MASK_29BIT;
ht_Compressor_Status.Data[0]	:=	16#FF;
ht_Compressor_Status.Data[1]	:=	16#FF;
ht_Compressor_Status.Data[2]	:=	16#FF;
ht_Compressor_Status.Data[3]	:=	16#FF;
ht_Compressor_Status.Data[4]	:=	16#FF;
ht_Compressor_Status.Data[5]	:=	16#FF;
ht_Compressor_Status.Data[6].0	:=	gq_Merc_AirComp_Enabled;
ht_Compressor_Status.Data[6].1	:=	0;
ht_Compressor_Status.Data[6].2	:=	1;
ht_Compressor_Status.Data[6].3	:=	1;
ht_Compressor_Status.Data[6].4	:=	1;
ht_Compressor_Status.Data[6].5	:=	1;
ht_Compressor_Status.Data[6].6	:=	1;
ht_Compressor_Status.Data[6].7	:=	1;
ht_Compressor_Status.Data[7]	:=	16#FF;
ht_Compressor_Status.Len	:=	8;*)


(*10ms*)
hu8_4BitMessageCounter10ms	:=	hu8_4BitMessageCounter10ms + 1;
IF (hu8_4BitMessageCounter10ms > 15) THEN
	hu8_4BitMessageCounter10ms	:=	0;
END_IF
G_CAN1_Channel.SendMessage(i_pMSG:=ADR(ht_TCM_C01_Tx));
G_CAN1_Channel.SendMessage(i_pMSG:=ADR(ht_TCM_C02_Tx));
G_CAN1_Channel.SendMessage(i_pMSG:=ADR(ht_TCM_C03_Tx));
G_CAN1_Channel.SendMessage(i_pMSG:=ADR(ht_TCM_C11_Tx));
G_CAN1_Channel.SendMessage(i_pMSG:=ADR(ht_MCM_C01_Tx));
G_CAN1_Channel.SendMessage(i_pMSG:=ADR(ht_MCM_C02_Tx));
G_CAN1_Channel.SendMessage(i_pMSG:=ADR(ht_MCM_C23_Tx));

IF (hq_CycleAlternator = TRUE) THEN
	hu8_4BitMessageCounter20ms	:=	hu8_4BitMessageCounter20ms + 1;
	IF (hu8_4BitMessageCounter20ms > 15) THEN
		hu8_4BitMessageCounter20ms	:=	0;
	END_IF
	G_CAN1_Channel.SendMessage(i_pMSG:=ADR(ht_RCM_C01_Tx));
	G_CAN1_Channel.SendMessage(i_pMSG:=ADR(ht_TCM_C08_Tx));
	G_CAN1_Channel.SendMessage(i_pMSG:=ADR(ht_MCM_C15_Tx));
END_IF
hq_CycleAlternator	:=	NOT(hq_CycleAlternator);

hton_MessageSend50ms_Timer(IN := NOT(hton_MessageSend50ms_Timer.Q), PT := T#50MS);
IF (hton_MessageSend50ms_Timer.Q = TRUE) THEN
	hu8_4BitMessageCounter50ms	:=	hu8_4BitMessageCounter50ms + 1;
	IF (hu8_4BitMessageCounter50ms > 15) THEN
		hu8_4BitMessageCounter50ms	:=	0;
	END_IF
	G_CAN1_Channel.SendMessage(i_pMSG:=ADR(ht_TCM_C10_Tx));
END_IF

hton_MessageSend_Timer(IN := NOT(hton_MessageSend_Timer.Q), PT := T#100MS);
IF (hton_MessageSend_Timer.Q = TRUE) THEN	
	hu8_4BitMessageCounter100ms	:=	hu8_4BitMessageCounter100ms + 1;
	IF (hu8_4BitMessageCounter100ms > 15) THEN
		hu8_4BitMessageCounter100ms	:=	0;
	END_IF
	G_CAN1_Channel.SendMessage(i_pMSG:=ADR(ht_RCM_C02_Tx));
	G_CAN1_Channel.SendMessage(i_pMSG:=ADR(ht_TCM_C05_Tx));
	G_CAN1_Channel.SendMessage(i_pMSG:=ADR(ht_MCM_C03_Tx));
	G_CAN1_Channel.SendMessage(i_pMSG:=ADR(ht_MCM_C07_Tx));
END_IF

Tx_Timer(IN := NOT(Tx_Timer.Q), PT := T#1000MS);
IF (Tx_Timer.Q = TRUE) THEN
	G_CAN1_Channel.SendMessage(i_pMSG:=ADR(ht_TCM_C06_Tx));
	G_CAN1_Channel.SendMessage(i_pMSG:=ADR(ht_TCM_C22_Tx));
	G_CAN1_Channel.SendMessage(i_pMSG:=ADR(ht_TRF1_TCM_Tx));
	G_CAN1_Channel.SendMessage(i_pMSG:=ADR(ht_MCM_C10_Tx));
	G_CAN1_Channel.SendMessage(i_pMSG:=ADR(ht_MCM_C14_Tx));
	
	G_CAN1_Channel.SendMessage(i_pMSG:=ADR(ht_Compressor_Status));
	
END_IF

(* Below is to alter the state of the clutch *)
IF gq_Merc_Neutral = TRUE THEN
	ClutchStatA := FALSE;
	ClutchStatB := TRUE;
	ClutchDisengaged := TRUE;
ELSE 
	ClutchDisengaged := FALSE;
END_IF

IF 	(gq_Merc_Drive OR gq_Merc_Reverse = TRUE) AND gq_BrakeSwitch THEN
	ClutchStatA := TRUE;
	ClutchStatB := FALSE;
	ClutchIntermediate := TRUE;
ELSE
	ClutchIntermediate := FALSE;
END_IF

IF (ClutchIntermediate = TRUE) THEN
	TONIntermediate (IN := TRUE, PT := T#50MS);
ELSIF (gq_Merc_Neutral = TRUE) THEN
	TONIntermediate (IN := FALSE, PT := T#0MS);
END_IF

IF 	(gq_Merc_Drive OR gq_Merc_Reverse = TRUE) AND 
	(TONIntermediate.Q = TRUE) THEN
	ClutchStatA := FALSE;
	ClutchStatB := FALSE;
	ClutchEngaged := TRUE;
ELSE
	ClutchEngaged := FALSE;
END_IF

END_PROGRAM

// GetLibVersion
// This function has been automatically generated from the project information.
FUNCTION GetLibVersion : VERSION
VAR_INPUT
	
END_VAR

GetLibVersion.uiMajor := 3;
GetLibVersion.uiMinor := 0;
GetLibVersion.uiServicePack := 6;
GetLibVersion.uiPatch := 65535;

END_FUNCTION

// GetLibVersionNumber
// This function has been automatically generated from the project information.
FUNCTION GetLibVersionNumber : DWORD
VAR_INPUT
	
END_VAR

GetLibVersionNumber := 50333439;

END_FUNCTION

// IsLibReleased
// This function has been automatically generated from the project information.
FUNCTION IsLibReleased : BOOL
VAR_INPUT
	
END_VAR

IsLibReleased := FALSE;

END_FUNCTION

// GetBooleanProperty
// This function has been automatically generated from the project information.
{attribute 'signature_flag' := '1073741824'}
{attribute 'register_in_runtime'}
FUNCTION GetBooleanProperty : BOOL
VAR_INPUT
	stKey: WSTRING;
END_VAR

GetBooleanProperty := FALSE;

END_FUNCTION

// GetCompany
// This function has been automatically generated from the project information.
{attribute 'signature_flag' := '1073741824'}
{attribute 'register_in_runtime'}
FUNCTION GetCompany : WSTRING
VAR_INPUT
	
END_VAR

GetCompany := "Electra";

END_FUNCTION

// GetNumberProperty
// This function has been automatically generated from the project information.
{attribute 'signature_flag' := '1073741824'}
{attribute 'register_in_runtime'}
FUNCTION GetNumberProperty : DINT
VAR_INPUT
	stKey: WSTRING;
END_VAR

GetNumberProperty := 0;

END_FUNCTION

// GetTextProperty2
// This function has been automatically generated from the project information.
{attribute 'signature_flag' := '1073741824'}
{attribute 'register_in_runtime'}
FUNCTION GetTextProperty2 : POINTER TO WSTRING
VAR_INPUT
	stKey: WSTRING;
END_VAR

IF stKey = "Author" THEN
	GetTextProperty2 := ADR("Luke");
ELSIF stKey = "Company" THEN
	GetTextProperty2 := ADR("Electra");
ELSIF stKey = "CompiledLibraryCompatibilityVersion" THEN
	GetTextProperty2 := ADR("CODESYS V3.5 SP13");
ELSIF stKey = "Description" THEN
	GetTextProperty2 := ADR("Reduced Brusa Temps for fan
ePTO set to activate with reverse
Cooling Fan reinstated
Additional compressor run signals
Gear change adjustment
Comp temp Error SP raised
Auto regen on overspeed >56@5s
OR t AND for Traction Off Keypad Combo
");
ELSIF stKey = "Project" THEN
	GetTextProperty2 := ADR("e-Compact_3.0.6_FCC");
ELSIF stKey = "Title" THEN
	GetTextProperty2 := ADR("e-Compact");
ELSE
	GetTextProperty2 := ADR("");
END_IF

END_FUNCTION

// GetTextProperty
// This function has been automatically generated from the project information.
{attribute 'signature_flag' := '1073741824'}
{attribute 'register_in_runtime'}
FUNCTION GetTextProperty : WSTRING
VAR_INPUT
	stKey: WSTRING;
END_VAR

IF stKey = "Author" THEN
	GetTextProperty := "Luke";
ELSIF stKey = "Company" THEN
	GetTextProperty := "Electra";
ELSIF stKey = "CompiledLibraryCompatibilityVersion" THEN
	GetTextProperty := "CODESYS V3.5 SP13";
ELSIF stKey = "Description" THEN
	GetTextProperty := "Reduced Brusa Temps for fan
ePTO set to activate with reverse
Cooling Fan reinstated
Additional compressor run signals
Gear change adjustment
Comp temp Error SP raised
Auto regen on overspeed >56@5s
OR t AND for Traction Off Keypad Combo
";
ELSIF stKey = "Project" THEN
	GetTextProperty := "e-Compact_3.0.6_FCC";
ELSIF stKey = "Title" THEN
	GetTextProperty := "e-Compact";
ELSE
	GetTextProperty := "";
END_IF

END_FUNCTION

// GetTitle
// This function has been automatically generated from the project information.
{attribute 'signature_flag' := '1073741824'}
{attribute 'register_in_runtime'}
FUNCTION GetTitle : WSTRING
VAR_INPUT
	
END_VAR

GetTitle := "e-Compact";

END_FUNCTION

// GetVersion
// This function has been automatically generated from the project information.
{attribute 'signature_flag' := '1073741824'}
{attribute 'register_in_runtime'}
FUNCTION GetVersion : VERSION
VAR_INPUT
	
END_VAR

GetVersion.uiMajor := 3;
GetVersion.uiMinor := 0;
GetVersion.uiServicePack := 6;
GetVersion.uiPatch := 65535;

END_FUNCTION

// GetVersionProperty
// This function has been automatically generated from the project information.
{attribute 'signature_flag' := '1073741824'}
{attribute 'register_in_runtime'}
FUNCTION GetVersionProperty : VERSION
VAR_INPUT
	stKey: WSTRING;
END_VAR

IF stKey = "Version" THEN
	GetVersionProperty.uiMajor := 3;
	GetVersionProperty.uiMinor := 0;
	GetVersionProperty.uiServicePack := 6;
	GetVersionProperty.uiPatch := 65535;
ELSE
	GetVersionProperty.uiMajor := 0;
	GetVersionProperty.uiMinor := 0;
	GetVersionProperty.uiServicePack := 0;
	GetVersionProperty.uiPatch := 0;
END_IF

END_FUNCTION

// Application/UserCode/BELDCDC/BELDCDC_Control_1
PROGRAM BELDCDC_Control_1
VAR
	hton_DelayTimer	:	TON;
END_VAR

(*Setting the digital outputs to the DCDC*)

IF (DOS_q_BatteryDischargeMain_DO = TRUE AND gu8_SystemState = DRIVE_SYS) THEN
	(*Once the main contactor is connected wait 5 seconds then set the ouputs high*)
	hton_DelayTimer(IN := TRUE, PT := T#5S);
	DO_q_DrivetrainDCDCInhibit_DO	:=	hton_DelayTimer.Q;
	DO_q_DashboardDCDCStatus_DO		:=	hton_DelayTimer.Q;
ELSIF (DO_q_Battery1ChargeMain_DO = TRUE OR DO_q_Battery2ChargeMain_DO = TRUE) THEN
	(*Switch off outputs when in charge*)
	hton_DelayTimer(IN := FALSE, PT := T#0S);
	DO_q_DrivetrainDCDCInhibit_DO	:=	FALSE;
	DO_q_DashboardDCDCStatus_DO		:=	FALSE;
	(*This is included for future so that the DCDC can be brought in during charge but is not possible with current electrical setup*)
ELSE
	(*Any other state switch outputs off*)
	hton_DelayTimer(IN := FALSE, PT := T#0S);
	DO_q_DrivetrainDCDCInhibit_DO	:=	FALSE;
	DO_q_DashboardDCDCStatus_DO		:=	FALSE;
END_IF

END_PROGRAM

// Application/UserCode/BELDCDC/BELDCDC_Rx_1
PROGRAM BELDCDC_Rx_1
VAR
	BelDCDC_FWS_Rx			:	Receive_CAN1_EXD;
	BelDCDC_IO_Rx			:	Receive_CAN1_EXD;
	BelDCDC_FWS_Rx_Timer	:	TON;
	BelDCDC_IO_Rx_Timer		:	TON;
	hton_Startup_Timer		:	TON;
	Fault_InputUV			:	BOOL;
	Fault_InputOV			:	BOOL;
	Fault_OutputUV			:	BOOL;
	Fault_OutputOV			:	BOOL;
	Fault_OutputOC			:	BOOL;
	Fault_OTP				:	BOOL;
	Fault_I2CFault			:	BOOL;
	Fault_CANFault			:	BOOL;
	Fault_EEPROM_CRCFault	:	BOOL;
	Fault_ShortCircuit		:	BOOL;
	Fault_ThermistorFault	:	BOOL;
	Fault_Overload			:	BOOL;
	Fault_OutputOVLatch		:	BOOL;
	Fault_ReversePolarity	:	BOOL;
	Warning_CoolantOTP		:	BOOL;
	Warning_CurrentLimiting	:	BOOL;
	Status_UnitEnabled		:	BOOL;
	Status_Wakeup			:	BOOL;
	Status_Fault			:	BOOL;
	Status_LatchedFault		:	BOOL;
	Status_RemoteShutdown	:	BOOL;
	Status_StartupInitDone	:	BOOL;
	Status_InputOK			:	BOOL;
	Status_HVILOK			:	BOOL;
	Status_ReversePolarity	:	BOOL;
	Status_Hiccup			:	BOOL;
	OutputVoltage_Rx		:	UINT;
	OutputCurrent_Rx		:	UINT;
	InputVoltage_Rx			:	UINT;
	TempCoolant_Rx			:	UINT;
	CommsLoss				:	BOOL;
END_VAR

(*Message receipt for the DCDCs*)

(*Receive the messages from the DCDC*)
BelDCDC_FWS_Rx(u32_COBID	:=	16#18FFD4B3,
				 q_NewData => ,
				 au8_Data => ,
				 u8_Length => 			);

BelDCDC_IO_Rx(u32_COBID	:=	16#18FFD6B3,
				 q_NewData => ,
				 au8_Data => ,
				 u8_Length => 			);

(*Wait an initial time from when the DCDC is switched on to prevent falsly detecting faults*)
hton_Startup_Timer(IN := DO_q_DrivetrainDCDCInhibit_DO, PT := T#1000MS);
IF (hton_Startup_Timer.Q = TRUE) THEN (*During startup errors are reported while precharge occurs so this ignores the initiall error reporting*)
	Fault_InputUV			:=	BelDCDC_FWS_Rx.au8_Data[0].0;
	Fault_InputOV			:=	BelDCDC_FWS_Rx.au8_Data[0].1;
	Fault_OutputUV			:=	BelDCDC_FWS_Rx.au8_Data[0].2;
	Fault_OutputOV			:=	BelDCDC_FWS_Rx.au8_Data[0].3;
	Fault_OutputOC			:=	BelDCDC_FWS_Rx.au8_Data[0].4;
	Fault_OTP				:=	BelDCDC_FWS_Rx.au8_Data[0].5;
	Fault_I2CFault			:=	BelDCDC_FWS_Rx.au8_Data[0].6;
	Fault_CANFault			:=	BelDCDC_FWS_Rx.au8_Data[0].7;
	Fault_EEPROM_CRCFault	:=	BelDCDC_FWS_Rx.au8_Data[1].0;
	Fault_ShortCircuit		:=	BelDCDC_FWS_Rx.au8_Data[1].1;
	Fault_ThermistorFault	:=	BelDCDC_FWS_Rx.au8_Data[1].2;
	Fault_Overload			:=	BelDCDC_FWS_Rx.au8_Data[1].3;
	Fault_OutputOVLatch		:=	BelDCDC_FWS_Rx.au8_Data[1].4;
	Fault_ReversePolarity	:=	BelDCDC_FWS_Rx.au8_Data[1].5;
	Warning_CoolantOTP		:=	BelDCDC_FWS_Rx.au8_Data[3].0;
	Warning_CurrentLimiting	:=	BelDCDC_FWS_Rx.au8_Data[3].1;
	Status_UnitEnabled		:=	BelDCDC_FWS_Rx.au8_Data[6].0;
	Status_Wakeup			:=	BelDCDC_FWS_Rx.au8_Data[6].1;
	Status_Fault			:=	BelDCDC_FWS_Rx.au8_Data[6].2;
	Status_LatchedFault		:=	BelDCDC_FWS_Rx.au8_Data[6].3;
	Status_RemoteShutdown	:=	BelDCDC_FWS_Rx.au8_Data[6].4;
	Status_StartupInitDone	:=	BelDCDC_FWS_Rx.au8_Data[6].5;
	Status_InputOK			:=	BelDCDC_FWS_Rx.au8_Data[6].6;
	Status_HVILOK			:=	BelDCDC_FWS_Rx.au8_Data[6].7;
	Status_ReversePolarity	:=	BelDCDC_FWS_Rx.au8_Data[7].0;
	Status_Hiccup			:=	BelDCDC_FWS_Rx.au8_Data[7].1;
END_IF
(*IO*)
OutputVoltage_Rx			:=	USINT_TO_UINT(BelDCDC_IO_Rx.au8_Data[0]) +
									SHL(USINT_TO_UINT(BelDCDC_IO_Rx.au8_Data[1]), 8);
OutputCurrent_Rx			:=	USINT_TO_UINT(BelDCDC_IO_Rx.au8_Data[2]) +
									SHL(USINT_TO_UINT(BelDCDC_IO_Rx.au8_Data[3]), 8);
InputVoltage_Rx				:=	USINT_TO_UINT(BelDCDC_IO_Rx.au8_Data[4]) +
									SHL(USINT_TO_UINT(BelDCDC_IO_Rx.au8_Data[5]), 8);
TempCoolant_Rx				:=	USINT_TO_UINT(BelDCDC_IO_Rx.au8_Data[6]) +
									SHL(USINT_TO_UINT(BelDCDC_IO_Rx.au8_Data[7]), 8);

(*Bel DCDC only seems to send messages on startup*)
(*When the output is set then detect if messages are being sent if no message is received for 5 seconds then report a communications loss*)
BelDCDC_FWS_Rx_Timer(IN := (NOT(BelDCDC_FWS_Rx.q_NewData) AND DO_q_DrivetrainDCDCInhibit_DO = TRUE), PT := T#5S);
BelDCDC_IO_Rx_Timer(IN := (NOT(BelDCDC_IO_Rx.q_NewData) AND DO_q_DrivetrainDCDCInhibit_DO = TRUE), PT := T#5S);
IF (BelDCDC_FWS_Rx_Timer.Q = TRUE AND BelDCDC_IO_Rx_Timer.Q = TRUE) THEN
	CommsLoss	:=	TRUE;
ELSE
	CommsLoss	:=	FALSE;
END_IF									

BELDCDC_RxConversion();

END_PROGRAM

// Application/UserCode/BELDCDC/BELDCDC_RxConversion_1
PROGRAM BELDCDC_RxConversion_1
VAR
	OutputVoltage		:	REAL;
	OutputCurrent		:	REAL;
	InputVoltage		:	REAL;
	TempCoolant			:	REAL;
END_VAR

(*Take the values received on CANbus and apply the offset and conversion factor to each where necessary*)
OutputVoltage		:=	UINT_TO_REAL(BELDCDC_Rx.OutputVoltage_Rx) * 0.05;
OutputCurrent		:=	UINT_TO_REAL(BELDCDC_Rx.OutputCurrent_Rx) * 0.05;
InputVoltage			:=	UINT_TO_REAL(BELDCDC_Rx.InputVoltage_Rx) * 0.05;
TempCoolant			:=	UINT_TO_REAL(BELDCDC_Rx.TempCoolant_Rx) * 0.1;

END_PROGRAM

// Application/UserCode/BELDCDC/BELDCDC_Tx_1
PROGRAM BELDCDC_Tx_1
VAR
	BelDCDC_TX				:	EPEC_CANVXD.Msg;
	hton_MessageSend_Timer	:	TON;
	DCDC_Enable: BYTE 		:= 1; // Enable Bit (There is also a HW wire)
END_VAR

(*Message Transmit for the DCDC*)
BelDCDC_TX.ID	:=	16#18EFB300 OR EPEC_CANVXD.MASK_29BIT;//* message to control DCDC
BelDCDC_TX.Data[0]	:=	0;//* system requirement.
BelDCDC_TX.Data[1]	:=	WORD_TO_BYTE (BELDCDC_TxConversion.RAW_DCDC_Voltage_SP);//*LSB
BelDCDC_TX.Data[2]	:=	WORD_TO_BYTE (SHR (BELDCDC_TxConversion.RAW_DCDC_Voltage_SP,8));//*MSB
BelDCDC_TX.Data[3]	:=	WORD_TO_BYTE (BELDCDC_TxConversion.RAW_DCDC_Current_SP);//*LSB
BelDCDC_TX.Data[4]	:=	WORD_TO_BYTE (SHR (BELDCDC_TxConversion.RAW_DCDC_Current_SP,8));//*MSB
BelDCDC_TX.Data[5]	:=	DCDC_Enable;
BelDCDC_TX.Data[6]	:=	255;//* system requirement.
BelDCDC_TX.Data[7]	:=	255;//* system requirement.
BelDCDC_TX.Len		:=	8;


hton_MessageSend_Timer(IN := NOT(hton_MessageSend_Timer.Q), PT := T#200MS);//* Tx every 200ms
IF (hton_MessageSend_Timer.Q = TRUE) THEN
G_CAN1_Channel.SendMessage(i_pMSG:=ADR(BelDCDC_TX));
END_IF

END_PROGRAM

// Application/UserCode/BELDCDC/BELDCDC_TxConversion_1
PROGRAM BELDCDC_TxConversion_1
VAR
	RAW_DCDC_Voltage_SP	: WORD;
	RAW_DCDC_Current_SP	: WORD;
	DCDC_Current_SP		: REAL := 100; // Amperage
	DCDC_Voltage_SP		: REAL :=27.6;// Battery Voltage	
END_VAR

(*Take the values and Tx over CANbus and apply the offset and conversion factor to each where necessary*)

RAW_DCDC_Voltage_SP					:=REAL_TO_WORD(DCDC_Voltage_SP*20);
RAW_DCDC_Current_SP					:=REAL_TO_WORD (DCDC_Current_SP*20);

END_PROGRAM

// Application/UserCode/BMS/BMSData_1
PROGRAM BMSData_1
VAR
	Batteries_Fully_Charged : BOOL;
	chargeInterlockFlt      : BOOL;
END_VAR


IF (gu8_BMS_SOC >= 100 AND gs16_BMS2_CCL <= 0 AND gs16_BMS1_CCL <= 0) THEN
	Batteries_Fully_Charged				:=	TRUE;
ELSE
	Batteries_Fully_Charged				:=	FALSE;
END_IF

CASE gu8_BMSType OF
	BMS_ORION:
		gu8_BMS_SOC						:=	REAL_TO_USINT (MIN(OrionBMS1_RxConversion.gr_OrionBMS1_PackSOC, OrionBMS2_RxConversion.gr_OrionBMS2_PackSOC));
		gr_BMS_BatteryVoltage			:=	REAL_TO_UINT((OrionBMS1_RxConversion.gr_OrionBMS1_PackVoltage + OrionBMS2_RxConversion.gr_OrionBMS2_PackVoltage));
		gr_BMS1_Voltage					:=	REAL_TO_UINT(OrionBMS1_RxConversion.gr_OrionBMS1_PackVoltage);
		gr_BMS2_Voltage					:=	REAL_TO_UINT(OrionBMS2_RxConversion.gr_OrionBMS2_PackVoltage);
		gs16_BMS_BatteryCurrent			:=	REAL_TO_INT((OrionBMS1_RxConversion.gr_OrionBMS1_PackCurrent + OrionBMS2_RxConversion.gr_OrionBMS2_PackCurrent) / 2);
		gu16_BMS_Maximum_Pack_Voltage	:=	REAL_TO_UINT(gu16_OrionBMS1_MaximumPackVoltage + gu16_OrionBMS2_MaximumPackVoltage) / 10; (*Limit applied to prevent overcharging*)
		gs16_BMS1_CCL					:=	UINT_TO_INT(gu16_OrionBMS1_PackCCL);
		gs16_BMS2_CCL					:=	UINT_TO_INT(gu16_OrionBMS2_PackCCL);
		gu16_BMS_AverageCellVoltage		:=	(gu16_OrionBMS1_AverageCellVoltage + gu16_OrionBMS2_AverageCellVoltage) / 2;
		gu16_BMS_LowCellVoltage			:=	MIN(gu16_OrionBMS1_LowCellVoltage, gu16_OrionBMS2_LowCellVoltage);
		gu16_BMS_HighCellVoltage		:=	MAX(gu16_OrionBMS1_HighCellVoltage, gu16_OrionBMS2_HighCellVoltage);
		gr_BMS_AverageTemp				:=	(gu8_OrionBMS1_AverageTemp + gu8_OrionBMS2_AverageTemp) / 2;
		gr_BMS_LowTemp					:=	MIN(gu8_OrionBMS1_LowTemp, gu8_OrionBMS2_LowTemp);
		gr_BMS_HighTemp					:=	MAX(gu8_OrionBMS1_HighTemp, gu8_OrionBMS2_HighTemp);
		gr_BMS_DCL						:=	MIN(gu16_OrionBMS1_PackDCL, gu16_OrionBMS2_PackDCL);
		gr_BMS_CCL						:=	MIN(gu16_OrionBMS1_PackCCL, gu16_OrionBMS2_PackCCL);
		gu16_BMS_MinimumPackVoltage		:=	(gu16_OrionBMS1_MinimumPackVoltage + gu16_OrionBMS2_MinimumPackVoltage) / 10;
		gu16_BMS1_LowCellVoltage		:=	gu16_OrionBMS1_LowCellVoltage;
		gu16_BMS2_LowCellVoltage		:=	gu16_OrionBMS2_LowCellVoltage;
		gu16_BMS1_HighCellVoltage		:=	gu16_OrionBMS1_HighCellVoltage;
		gu16_BMS2_HighCellVoltage		:=	gu16_OrionBMS2_HighCellVoltage;
		gu16_BMS1_LowCellVoltage_ID		:=	gu8_OrionBMS1_LowCellVoltNumber;
		gu16_BMS2_LowCellVoltage_ID		:=	gu8_OrionBMS2_LowCellVoltNumber;
		gu16_BMS1_HighCellVoltage_ID	:=	gu8_OrionBMS1_HighCellVoltNumber;
		gu16_BMS2_HighCellVoltage_ID	:=	gu8_OrionBMS2_HighCellVoltNumber;
		
		
